LIN {X 0,Y 523.92,Z 267.852,A -85,B 0,C 180,E1 -4812.457,E2 -4812.457} C_VEL
LIN {X 0,Y 523.943,Z 267.84,A -85,B 0,C 180,E1 -4815.311,E2 -4815.311} C_VEL
LIN {X 0,Y 523.959,Z 267.843,A -85,B 0,C 180,E1 -4818.69,E2 -4818.69} C_VEL
LIN {X 0,Y 523.916,Z 267.847,A -85,B 0,C 180,E1 -4821.898,E2 -4821.898} C_VEL
LIN {X 0,Y 523.925,Z 267.843,A -85,B 0,C 180,E1 -4824.912,E2 -4824.912} C_VEL
LIN {X 0,Y 523.939,Z 267.841,A -85,B 0,C 180,E1 -4827.68,E2 -4827.68} C_VEL
LIN {X 0,Y 523.957,Z 267.84,A -85,B 0,C 180,E1 -4830.677,E2 -4830.677} C_VEL
LIN {X 0,Y 523.932,Z 267.843,A -85,B 0,C 180,E1 -4833.726,E2 -4833.726} C_VEL
LIN {X 0,Y 523.915,Z 267.849,A -85,B 0,C 180,E1 -4836.27,E2 -4836.27} C_VEL
LIN {X 0,Y 523.95,Z 267.841,A -85,B 0,C 180,E1 -4838.767,E2 -4838.767} C_VEL
LIN {X 0,Y 523.942,Z 267.839,A -85,B 0,C 180,E1 -4841.22,E2 -4841.22} C_VEL
LIN {X 0,Y 523.926,Z 267.846,A -85,B 0,C 180,E1 -4843.639,E2 -4843.639} C_VEL
LIN {X 0,Y 523.939,Z 267.849,A -85,B 0,C 180,E1 -4846.028,E2 -4846.028} C_VEL
LIN {X 0,Y 523.996,Z 267.832,A -85,B 0,C 180,E1 -4849.177,E2 -4849.177} C_VEL
LIN {X 0,Y 523.96,Z 267.842,A -85,B 0,C 180,E1 -4851.515,E2 -4851.515} C_VEL
LIN {X 0,Y 524.041,Z 267.829,A -85,B 0,C 180,E1 -4854.613,E2 -4854.613} C_VEL
LIN {X 0,Y 524.107,Z 267.825,A -85,B 0,C 180,E1 -4857.695,E2 -4857.695} C_VEL
LIN {X 0,Y 524.1,Z 267.827,A -85,B 0,C 180,E1 -4860,E2 -4860} C_VEL
LIN {X 0,Y 524.037,Z 267.829,A -85,B 0,C 180,E1 -4863.075,E2 -4863.075} C_VEL
LIN {X 0,Y 524.002,Z 267.835,A -85,B 0,C 180,E1 -4866.16,E2 -4866.16} C_VEL
LIN {X 0,Y 523.948,Z 267.843,A -85,B 0,C 180,E1 -4869.263,E2 -4869.263} C_VEL
LIN {X 0,Y 524.001,Z 267.841,A -85,B 0,C 180,E1 -4871.735,E2 -4871.735} C_VEL
LIN {X 0,Y 523.987,Z 267.834,A -85,B 0,C 180,E1 -4875.047,E2 -4875.047} C_VEL
LIN {X 0,Y 523.914,Z 267.846,A -85,B 0,C 180,E1 -4877.971,E2 -4877.971} C_VEL
LIN {X 0,Y 523.92,Z 267.844,A -85,B 0,C 180,E1 -4880.412,E2 -4880.412} C_VEL
LIN {X 0,Y 523.888,Z 267.846,A -85,B 0,C 180,E1 -4882.895,E2 -4882.895} C_VEL
LIN {X 0,Y 523.883,Z 267.856,A -85,B 0,C 180,E1 -4885.422,E2 -4885.422} C_VEL
LIN {X 0,Y 523.9,Z 267.841,A -85,B 0,C 180,E1 -4888.003,E2 -4888.003} C_VEL
LIN {X 0,Y 523.901,Z 267.847,A -85,B 0,C 180,E1 -4890.845,E2 -4890.845} C_VEL
LIN {X 0,Y 523.914,Z 267.849,A -85,B 0,C 180,E1 -4893.726,E2 -4893.726} C_VEL
LIN {X 0,Y 523.86,Z 267.85,A -85,B 0,C 180,E1 -4896.394,E2 -4896.394} C_VEL
LIN {X 0,Y 523.889,Z 267.852,A -85,B 0,C 180,E1 -4899.088,E2 -4899.088} C_VEL
LIN {X 0,Y 523.888,Z 267.847,A -85,B 0,C 180,E1 -4902.125,E2 -4902.125} C_VEL
LIN {X 0,Y 523.927,Z 267.844,A -85,B 0,C 180,E1 -4904.687,E2 -4904.687} C_VEL
LIN {X 0,Y 523.857,Z 267.853,A -85,B 0,C 180,E1 -4906.864,E2 -4906.864} C_VEL
LIN {X 0,Y 523.17,Z 267.942,A -85,B 0,C 180,E1 -4907.506,E2 -4907.506} C_VEL
LIN {X 0,Y 520.306,Z 268.294,A -85,B 0,C 180,E1 -4908.547,E2 -4908.547} C_VEL
LIN {X 0,Y 517.908,Z 268.599,A -85,B 0,C 180,E1 -4909.386,E2 -4909.386} C_VEL
LIN {X 0,Y 516.896,Z 268.719,A -85,B 0,C 180,E1 -4910.034,E2 -4910.034} C_VEL
LIN {X 0,Y 516.822,Z 268.727,A -85,B 0,C 180,E1 -4910.253,E2 -4910.253} C_VEL
LIN {X 0,Y 516.798,Z 268.736,A -85,B 0,C 180,E1 -4913.247,E2 -4913.247} C_VEL
LIN {X 0,Y 516.868,Z 268.721,A -85,B 0,C 180,E1 -4916.117,E2 -4916.117} C_VEL
LIN {X 0,Y 516.85,Z 268.729,A -85,B 0,C 180,E1 -4918.944,E2 -4918.944} C_VEL
LIN {X 0,Y 516.857,Z 268.725,A -85,B 0,C 180,E1 -4922.11,E2 -4922.11} C_VEL
LIN {X 0,Y 516.831,Z 268.735,A -85,B 0,C 180,E1 -4925.067,E2 -4925.067} C_VEL
LIN {X 0,Y 516.903,Z 268.891,A -85,B 0,C 180,E1 -4925.606,E2 -4925.606} C_VEL
LIN {X 0,Y 518.761,Z 277.486,A -85,B 0,C 180,E1 -4927.108,E2 -4927.108} C_VEL
LIN {X 0,Y 518.929,Z 282.515,A -85,B 0,C 180,E1 -4927.924,E2 -4927.924} C_VEL
LIN {X 0,Y 518.898,Z 284.871,A -85,B 0,C 180,E1 -4928.27,E2 -4928.27} C_VEL
LIN {X 0,Y 521.958,Z 298.303,A -85,B 0,C 180,E1 -4928.601,E2 -4928.601} C_VEL
LIN {X 0,Y 520.969,Z 446.051,A -85,B 0,C 180,E1 -4930.702,E2 -4930.702} C_VEL
LIN {X 0,Y 520.739,Z 460.824,A -85,B 0,C 180,E1 -4931.027,E2 -4931.027} C_VEL
LIN {X 0,Y 520.374,Z 475.321,A -85,B 0,C 180,E1 -4931.495,E2 -4931.495} C_VEL
LIN {X 0,Y 519.924,Z 489.139,A -85,B 0,C 180,E1 -4932.09,E2 -4932.09} C_VEL
LIN {X 0,Y 519.531,Z 501.957,A -85,B 0,C 180,E1 -4932.787,E2 -4932.787} C_VEL
LIN {X 0,Y 518.971,Z 515.318,A -85,B 0,C 180,E1 -4933.68,E2 -4933.68} C_VEL
LIN {X 0,Y 518.458,Z 527.648,A -85,B 0,C 180,E1 -4934.682,E2 -4934.682} C_VEL
LIN {X 0,Y 517.945,Z 539.712,A -85,B 0,C 180,E1 -4935.863,E2 -4935.863} C_VEL
LIN {X 0,Y 517.493,Z 549.881,A -85,B 0,C 180,E1 -4937.051,E2 -4937.051} C_VEL
LIN {X 0,Y 517.092,Z 559.832,A -85,B 0,C 180,E1 -4938.435,E2 -4938.435} C_VEL
LIN {X 0,Y 516.786,Z 568.082,A -85,B 0,C 180,E1 -4939.817,E2 -4939.817} C_VEL
LIN {X 0,Y 516.576,Z 575.827,A -85,B 0,C 180,E1 -4941.393,E2 -4941.393} C_VEL
LIN {X 0,Y 516.431,Z 581.994,A -85,B 0,C 180,E1 -4942.964,E2 -4942.964} C_VEL
LIN {X 0,Y 516.377,Z 586.756,A -85,B 0,C 180,E1 -4944.533,E2 -4944.533} C_VEL
LIN {X 0,Y 516.326,Z 590.248,A -85,B 0,C 180,E1 -4946.097,E2 -4946.097} C_VEL
LIN {X 0,Y 516.258,Z 592.562,A -85,B 0,C 180,E1 -4947.659,E2 -4947.659} C_VEL
LIN {X 0,Y 516.156,Z 593.75,A -85,B 0,C 180,E1 -4949.219,E2 -4949.219} C_VEL
LIN {X 0,Y 516.157,Z 593.769,A -85,B 0,C 180,E1 -4950.78,E2 -4950.78} C_VEL
LIN {X 0,Y 516.259,Z 592.657,A -85,B 0,C 180,E1 -4952.34,E2 -4952.34} C_VEL
LIN {X 0,Y 516.326,Z 590.419,A -85,B 0,C 180,E1 -4953.902,E2 -4953.902} C_VEL
LIN {X 0,Y 516.373,Z 586.999,A -85,B 0,C 180,E1 -4955.467,E2 -4955.467} C_VEL
LIN {X 0,Y 516.429,Z 582.315,A -85,B 0,C 180,E1 -4957.035,E2 -4957.035} C_VEL
LIN {X 0,Y 516.573,Z 576.243,A -85,B 0,C 180,E1 -4958.607,E2 -4958.607} C_VEL
LIN {X 0,Y 516.776,Z 568.595,A -85,B 0,C 180,E1 -4960.183,E2 -4960.183} C_VEL
LIN {X 0,Y 517.069,Z 560.435,A -85,B 0,C 180,E1 -4961.565,E2 -4961.565} C_VEL
LIN {X 0,Y 517.471,Z 550.604,A -85,B 0,C 180,E1 -4962.949,E2 -4962.949} C_VEL
LIN {X 0,Y 517.892,Z 540.518,A -85,B 0,C 180,E1 -4964.138,E2 -4964.138} C_VEL
LIN {X 0,Y 518.371,Z 528.692,A -85,B 0,C 180,E1 -4965.312,E2 -4965.312} C_VEL
LIN {X 0,Y 518.996,Z 515.308,A -85,B 0,C 180,E1 -4966.41,E2 -4966.41} C_VEL
LIN {X 0,Y 519.562,Z 501.798,A -85,B 0,C 180,E1 -4967.313,E2 -4967.313} C_VEL
LIN {X 0,Y 520.023,Z 486.91,A -85,B 0,C 180,E1 -4968.11,E2 -4968.11} C_VEL
LIN {X 0,Y 520.477,Z 471.674,A -85,B 0,C 180,E1 -4968.73,E2 -4968.73} C_VEL
LIN {X 0,Y 520.782,Z 456.381,A -85,B 0,C 180,E1 -4969.181,E2 -4969.181} C_VEL
LIN {X 0,Y 521.016,Z 441.647,A -85,B 0,C 180,E1 -4969.46,E2 -4969.46} C_VEL
LIN {X 0,Y 522.012,Z 299.314,A -85,B 0,C 180,E1 -4971.472,E2 -4971.472} C_VEL
LIN {X 0,Y 520.274,Z 290.511,A -85,B 0,C 180,E1 -4971.676,E2 -4971.676} C_VEL
LIN {X 0,Y 518.874,Z 284.647,A -85,B 0,C 180,E1 -4971.83,E2 -4971.83} C_VEL
LIN {X 0,Y 519.035,Z 279.823,A -85,B 0,C 180,E1 -4972.592,E2 -4972.592} C_VEL
LIN {X 0,Y 517.73,Z 272.676,A -85,B 0,C 180,E1 -4973.818,E2 -4973.818} C_VEL
LIN {X 0,Y 516.884,Z 268.728,A -85,B 0,C 180,E1 -4974.516,E2 -4974.516} C_VEL
LIN {X 0,Y 516.867,Z 268.727,A -85,B 0,C 180,E1 -4977.536,E2 -4977.536} C_VEL
LIN {X 0,Y 516.844,Z 268.729,A -85,B 0,C 180,E1 -4980.207,E2 -4980.207} C_VEL
LIN {X 0,Y 516.858,Z 268.731,A -85,B 0,C 180,E1 -4982.949,E2 -4982.949} C_VEL
LIN {X 0,Y 516.817,Z 268.728,A -85,B 0,C 180,E1 -4985.784,E2 -4985.784} C_VEL
LIN {X 0,Y 516.869,Z 268.73,A -85,B 0,C 180,E1 -4988.717,E2 -4988.717} C_VEL
LIN {X 0,Y 516.841,Z 268.726,A -85,B 0,C 180,E1 -4991.782,E2 -4991.782} C_VEL
LIN {X 0,Y 516.894,Z 268.725,A -85,B 0,C 180,E1 -4995.007,E2 -4995.007} C_VEL
LIN {X 0,Y 516.827,Z 268.725,A -85,B 0,C 180,E1 -4998.409,E2 -4998.409} C_VEL
LIN {X 0,Y 516.851,Z 268.725,A -85,B 0,C 180,E1 -5001.281,E2 -5001.281} C_VEL
LIN {X 0,Y 516.824,Z 268.727,A -85,B 0,C 180,E1 -5004.677,E2 -5004.677} C_VEL
LIN {X 0,Y 516.862,Z 268.723,A -85,B 0,C 180,E1 -5007.462,E2 -5007.462} C_VEL
LIN {X 0,Y 516.836,Z 268.733,A -85,B 0,C 180,E1 -5010.491,E2 -5010.491} C_VEL
LIN {X 0,Y 516.83,Z 268.726,A -85,B 0,C 180,E1 -5013.337,E2 -5013.337} C_VEL
LIN {X 0,Y 516.864,Z 268.724,A -85,B 0,C 180,E1 -5015.926,E2 -5015.926} C_VEL
LIN {X 0,Y 516.851,Z 268.732,A -85,B 0,C 180,E1 -5018.461,E2 -5018.461} C_VEL
LIN {X 0,Y 516.872,Z 268.721,A -85,B 0,C 180,E1 -5020.954,E2 -5020.954} C_VEL
LIN {X 0,Y 516.828,Z 268.727,A -85,B 0,C 180,E1 -5023.407,E2 -5023.407} C_VEL
LIN {X 0,Y 516.865,Z 268.722,A -85,B 0,C 180,E1 -5025.833,E2 -5025.833} C_VEL
LIN {X 0,Y 516.942,Z 268.713,A -85,B 0,C 180,E1 -5029.028,E2 -5029.028} C_VEL
LIN {X 0,Y 516.924,Z 268.719,A -85,B 0,C 180,E1 -5032.186,E2 -5032.186} C_VEL
LIN {X 0,Y 516.98,Z 268.711,A -85,B 0,C 180,E1 -5034.539,E2 -5034.539} C_VEL
LIN {X 0,Y 517.074,Z 268.697,A -85,B 0,C 180,E1 -5037.663,E2 -5037.663} C_VEL
LIN {X 0,Y 517.088,Z 268.692,A -85,B 0,C 180,E1 -5040.779,E2 -5040.779} C_VEL
LIN {X 0,Y 516.968,Z 268.709,A -85,B 0,C 180,E1 -5043.117,E2 -5043.117} C_VEL
LIN {X 0,Y 516.972,Z 268.714,A -85,B 0,C 180,E1 -5046.244,E2 -5046.244} C_VEL
LIN {X 0,Y 516.936,Z 268.714,A -85,B 0,C 180,E1 -5049.389,E2 -5049.389} C_VEL
LIN {X 0,Y 516.951,Z 268.714,A -85,B 0,C 180,E1 -5051.807,E2 -5051.807} C_VEL
LIN {X 0,Y 516.944,Z 268.71,A -85,B 0,C 180,E1 -5055.146,E2 -5055.146} C_VEL
LIN {X 0,Y 516.911,Z 268.721,A -85,B 0,C 180,E1 -5058.223,E2 -5058.223} C_VEL
LIN {X 0,Y 516.911,Z 268.717,A -85,B 0,C 180,E1 -5060.701,E2 -5060.701} C_VEL
LIN {X 0,Y 516.889,Z 268.717,A -85,B 0,C 180,E1 -5064.073,E2 -5064.073} C_VEL
LIN {X 0,Y 516.896,Z 268.716,A -85,B 0,C 180,E1 -5066.659,E2 -5066.659} C_VEL
LIN {X 0,Y 516.908,Z 268.722,A -85,B 0,C 180,E1 -5069.523,E2 -5069.523} C_VEL
LIN {X 0,Y 516.894,Z 268.715,A -85,B 0,C 180,E1 -5072.543,E2 -5072.543} C_VEL
LIN {X 0,Y 516.87,Z 268.725,A -85,B 0,C 180,E1 -5075.33,E2 -5075.33} C_VEL
LIN {X 0,Y 516.878,Z 268.723,A -85,B 0,C 180,E1 -5077.943,E2 -5077.943} C_VEL
LIN {X 0,Y 516.881,Z 268.72,A -85,B 0,C 180,E1 -5080.742,E2 -5080.742} C_VEL
LIN {X 0,Y 516.881,Z 268.721,A -85,B 0,C 180,E1 -5082.832,E2 -5082.832} C_VEL
LIN {X 0,Y 516.893,Z 268.72,A -85,B 0,C 180,E1 -5085.007,E2 -5085.007} C_VEL
LIN {X 0,Y 516.912,Z 268.716,A -85,B 0,C 180,E1 -5088.399,E2 -5088.399} C_VEL
LIN {X 0,Y 516.879,Z 268.726,A -85,B 0,C 180,E1 -5091.284,E2 -5091.284} C_VEL
LIN {X 0,Y 516.887,Z 268.722,A -85,B 0,C 180,E1 -5094.221,E2 -5094.221} C_VEL
LIN {X 0,Y 516.894,Z 268.723,A -85,B 0,C 180,E1 -5097.053,E2 -5097.053} C_VEL
LIN {X 0,Y 516.891,Z 268.727,A -85,B 0,C 180,E1 -5099.797,E2 -5099.797} C_VEL
LIN {X 0,Y 516.928,Z 268.855,A -85,B 0,C 180,E1 -5101.281,E2 -5101.281} C_VEL
LIN {X 0,Y 520.068,Z 282.653,A -85,B 0,C 180,E1 -5103.315,E2 -5103.315} C_VEL
LIN {X 0,Y 519.444,Z 305.178,A -85,B 0,C 180,E1 -5106.265,E2 -5106.265} C_VEL
LIN {X 0,Y 518.893,Z 320.181,A -85,B 0,C 180,E1 -5108.197,E2 -5108.197} C_VEL
LIN {X 0,Y 521.904,Z 335.969,A -85,B 0,C 180,E1 -5108.563,E2 -5108.563} C_VEL
LIN {X 0,Y 520.836,Z 485.958,A -85,B 0,C 180,E1 -5110.694,E2 -5110.694} C_VEL
LIN {X 0,Y 520.575,Z 500.684,A -85,B 0,C 180,E1 -5111.042,E2 -5111.042} C_VEL
LIN {X 0,Y 520.166,Z 514.057,A -85,B 0,C 180,E1 -5111.488,E2 -5111.488} C_VEL
LIN {X 0,Y 519.693,Z 527.714,A -85,B 0,C 180,E1 -5112.082,E2 -5112.082} C_VEL
LIN {X 0,Y 519.218,Z 542.063,A -85,B 0,C 180,E1 -5112.879,E2 -5112.879} C_VEL
LIN {X 0,Y 518.679,Z 555.131,A -85,B 0,C 180,E1 -5113.772,E2 -5113.772} C_VEL
LIN {X 0,Y 518.225,Z 566.573,A -85,B 0,C 180,E1 -5114.708,E2 -5114.708} C_VEL
LIN {X 0,Y 517.747,Z 578.379,A -85,B 0,C 180,E1 -5115.858,E2 -5115.858} C_VEL
LIN {X 0,Y 517.359,Z 588.67,A -85,B 0,C 180,E1 -5117.048,E2 -5117.048} C_VEL
LIN {X 0,Y 516.957,Z 598.75,A -85,B 0,C 180,E1 -5118.435,E2 -5118.435} C_VEL
LIN {X 0,Y 516.748,Z 607.095,A -85,B 0,C 180,E1 -5119.817,E2 -5119.817} C_VEL
LIN {X 0,Y 516.515,Z 614.951,A -85,B 0,C 180,E1 -5121.392,E2 -5121.392} C_VEL
LIN {X 0,Y 516.391,Z 621.202,A -85,B 0,C 180,E1 -5122.965,E2 -5122.965} C_VEL
LIN {X 0,Y 516.351,Z 626.04,A -85,B 0,C 180,E1 -5124.533,E2 -5124.533} C_VEL
LIN {X 0,Y 516.307,Z 629.583,A -85,B 0,C 180,E1 -5126.098,E2 -5126.098} C_VEL
LIN {X 0,Y 516.258,Z 631.912,A -85,B 0,C 180,E1 -5127.66,E2 -5127.66} C_VEL
LIN {X 0,Y 516.157,Z 633.082,A -85,B 0,C 180,E1 -5129.22,E2 -5129.22} C_VEL
LIN {X 0,Y 516.157,Z 633.081,A -85,B 0,C 180,E1 -5130.781,E2 -5130.781} C_VEL
LIN {X 0,Y 516.258,Z 631.908,A -85,B 0,C 180,E1 -5132.341,E2 -5132.341} C_VEL
LIN {X 0,Y 516.307,Z 629.577,A -85,B 0,C 180,E1 -5133.903,E2 -5133.903} C_VEL
LIN {X 0,Y 516.351,Z 626.039,A -85,B 0,C 180,E1 -5135.468,E2 -5135.468} C_VEL
LIN {X 0,Y 516.392,Z 621.204,A -85,B 0,C 180,E1 -5137.036,E2 -5137.036} C_VEL
LIN {X 0,Y 516.515,Z 614.944,A -85,B 0,C 180,E1 -5138.608,E2 -5138.608} C_VEL
LIN {X 0,Y 516.749,Z 607.085,A -85,B 0,C 180,E1 -5140.184,E2 -5140.184} C_VEL
LIN {X 0,Y 516.978,Z 598.727,A -85,B 0,C 180,E1 -5141.568,E2 -5141.568} C_VEL
LIN {X 0,Y 517.36,Z 588.664,A -85,B 0,C 180,E1 -5142.953,E2 -5142.953} C_VEL
LIN {X 0,Y 517.724,Z 578.372,A -85,B 0,C 180,E1 -5144.144,E2 -5144.144} C_VEL
LIN {X 0,Y 518.243,Z 566.539,A -85,B 0,C 180,E1 -5145.295,E2 -5145.295} C_VEL
LIN {X 0,Y 518.728,Z 553.828,A -85,B 0,C 180,E1 -5146.328,E2 -5146.328} C_VEL
LIN {X 0,Y 519.3,Z 540.456,A -85,B 0,C 180,E1 -5147.221,E2 -5147.221} C_VEL
LIN {X 0,Y 519.815,Z 525.705,A -85,B 0,C 180,E1 -5148.016,E2 -5148.016} C_VEL
LIN {X 0,Y 520.243,Z 511.445,A -85,B 0,C 180,E1 -5148.612,E2 -5148.612} C_VEL
LIN {X 0,Y 520.629,Z 495.966,A -85,B 0,C 180,E1 -5149.088,E2 -5149.088} C_VEL
LIN {X 0,Y 520.9,Z 480.134,A -85,B 0,C 180,E1 -5149.403,E2 -5149.403} C_VEL
LIN {X 0,Y 521.865,Z 335.63,A -85,B 0,C 180,E1 -5151.443,E2 -5151.443} C_VEL
LIN {X 0,Y 518.918,Z 320.204,A -85,B 0,C 180,E1 -5151.799,E2 -5151.799} C_VEL
LIN {X 0,Y 519.657,Z 297.1,A -85,B 0,C 180,E1 -5154.788,E2 -5154.788} C_VEL
LIN {X 0,Y 520.077,Z 282.636,A -85,B 0,C 180,E1 -5156.686,E2 -5156.686} C_VEL
LIN {X 0,Y 517.049,Z 269.454,A -85,B 0,C 180,E1 -5158.63,E2 -5158.63} C_VEL
LIN {X 0,Y 516.905,Z 268.725,A -85,B 0,C 180,E1 -5158.749,E2 -5158.749} C_VEL
LIN {X 0,Y 516.891,Z 268.723,A -85,B 0,C 180,E1 -5161.11,E2 -5161.11} C_VEL
LIN {X 0,Y 516.91,Z 268.721,A -85,B 0,C 180,E1 -5163.966,E2 -5163.966} C_VEL
LIN {X 0,Y 516.879,Z 268.726,A -85,B 0,C 180,E1 -5166.747,E2 -5166.747} C_VEL
LIN {X 0,Y 516.885,Z 268.718,A -85,B 0,C 180,E1 -5169.722,E2 -5169.722} C_VEL
LIN {X 0,Y 516.909,Z 268.718,A -85,B 0,C 180,E1 -5171.776,E2 -5171.776} C_VEL
LIN {X 0,Y 516.898,Z 268.72,A -85,B 0,C 180,E1 -5175.007,E2 -5175.007} C_VEL
LIN {X 0,Y 516.916,Z 268.725,A -85,B 0,C 180,E1 -5178.399,E2 -5178.399} C_VEL
LIN {X 0,Y 516.88,Z 268.721,A -85,B 0,C 180,E1 -5181.284,E2 -5181.284} C_VEL
LIN {X 0,Y 516.87,Z 268.729,A -85,B 0,C 180,E1 -5184.22,E2 -5184.22} C_VEL
LIN {X 0,Y 516.899,Z 268.717,A -85,B 0,C 180,E1 -5187.053,E2 -5187.053} C_VEL
LIN {X 0,Y 516.896,Z 268.721,A -85,B 0,C 180,E1 -5189.797,E2 -5189.797} C_VEL
LIN {X 0,Y 516.896,Z 268.722,A -85,B 0,C 180,E1 -5192.466,E2 -5192.466} C_VEL
LIN {X 0,Y 516.865,Z 268.722,A -85,B 0,C 180,E1 -5195.07,E2 -5195.07} C_VEL
LIN {X 0,Y 516.874,Z 268.721,A -85,B 0,C 180,E1 -5197.622,E2 -5197.622} C_VEL
LIN {X 0,Y 516.934,Z 268.72,A -85,B 0,C 180,E1 -5200.13,E2 -5200.13} C_VEL
LIN {X 0,Y 516.9,Z 268.72,A -85,B 0,C 180,E1 -5202.595,E2 -5202.595} C_VEL
LIN {X 0,Y 516.948,Z 268.71,A -85,B 0,C 180,E1 -5205.03,E2 -5205.03} C_VEL
LIN {X 0,Y 516.972,Z 268.712,A -85,B 0,C 180,E1 -5208.234,E2 -5208.234} C_VEL
LIN {X 0,Y 516.936,Z 268.716,A -85,B 0,C 180,E1 -5211.399,E2 -5211.399} C_VEL
LIN {X 0,Y 516.992,Z 268.708,A -85,B 0,C 180,E1 -5214.54,E2 -5214.54} C_VEL
LIN {X 0,Y 517.077,Z 268.7,A -85,B 0,C 180,E1 -5217.663,E2 -5217.663} C_VEL
LIN {X 0,Y 517.069,Z 268.703,A -85,B 0,C 180,E1 -5220,E2 -5220} C_VEL
LIN {X 0,Y 517.079,Z 268.697,A -85,B 0,C 180,E1 -5222.337,E2 -5222.337} C_VEL
LIN {X 0,Y 516.985,Z 268.712,A -85,B 0,C 180,E1 -5225.461,E2 -5225.461} C_VEL
LIN {X 0,Y 516.929,Z 268.715,A -85,B 0,C 180,E1 -5228.601,E2 -5228.601} C_VEL
LIN {X 0,Y 516.958,Z 268.718,A -85,B 0,C 180,E1 -5231.807,E2 -5231.807} C_VEL
LIN {X 0,Y 516.94,Z 268.712,A -85,B 0,C 180,E1 -5235.142,E2 -5235.142} C_VEL
LIN {X 0,Y 516.874,Z 268.72,A -85,B 0,C 180,E1 -5238.224,E2 -5238.224} C_VEL
LIN {X 0,Y 516.875,Z 268.721,A -85,B 0,C 180,E1 -5240.703,E2 -5240.703} C_VEL
LIN {X 0,Y 516.844,Z 268.727,A -85,B 0,C 180,E1 -5243.225,E2 -5243.225} C_VEL
LIN {X 0,Y 516.864,Z 268.721,A -85,B 0,C 180,E1 -5246.177,E2 -5246.177} C_VEL
LIN {X 0,Y 516.832,Z 268.719,A -85,B 0,C 180,E1 -5248.421,E2 -5248.421} C_VEL
LIN {X 0,Y 516.851,Z 268.728,A -85,B 0,C 180,E1 -5251.112,E2 -5251.112} C_VEL
LIN {X 0,Y 516.872,Z 268.724,A -85,B 0,C 180,E1 -5253.959,E2 -5253.959} C_VEL
LIN {X 0,Y 516.802,Z 268.73,A -85,B 0,C 180,E1 -5256.752,E2 -5256.752} C_VEL
LIN {X 0,Y 516.825,Z 268.731,A -85,B 0,C 180,E1 -5259.727,E2 -5259.727} C_VEL
LIN {X 0,Y 516.839,Z 268.728,A -85,B 0,C 180,E1 -5262.836,E2 -5262.836} C_VEL
LIN {X 0,Y 516.865,Z 268.727,A -85,B 0,C 180,E1 -5265.003,E2 -5265.003} C_VEL
LIN {X 0,Y 516.825,Z 268.727,A -85,B 0,C 180,E1 -5268.215,E2 -5268.215} C_VEL
LIN {X 0,Y 516.822,Z 268.727,A -85,B 0,C 180,E1 -5270.253,E2 -5270.253} C_VEL
LIN {X 0,Y 516.177,Z 268.814,A -85,B 0,C 180,E1 -5270.903,E2 -5270.903} C_VEL
LIN {X 0,Y 513.323,Z 269.17,A -85,B 0,C 180,E1 -5271.959,E2 -5271.959} C_VEL
LIN {X 0,Y 510.893,Z 269.474,A -85,B 0,C 180,E1 -5272.809,E2 -5272.809} C_VEL
LIN {X 0,Y 509.844,Z 269.603,A -85,B 0,C 180,E1 -5273.465,E2 -5273.465} C_VEL
LIN {X 0,Y 509.757,Z 269.611,A -85,B 0,C 180,E1 -5273.688,E2 -5273.688} C_VEL
LIN {X 0,Y 509.826,Z 269.6,A -85,B 0,C 180,E1 -5276.536,E2 -5276.536} C_VEL
LIN {X 0,Y 509.803,Z 269.61,A -85,B 0,C 180,E1 -5279.331,E2 -5279.331} C_VEL
LIN {X 0,Y 509.824,Z 269.602,A -85,B 0,C 180,E1 -5282.05,E2 -5282.05} C_VEL
LIN {X 0,Y 509.805,Z 269.611,A -85,B 0,C 180,E1 -5285.135,E2 -5285.135} C_VEL
LIN {X 0,Y 509.841,Z 269.786,A -85,B 0,C 180,E1 -5285.353,E2 -5285.353} C_VEL
LIN {X 0,Y 511.984,Z 279.585,A -85,B 0,C 180,E1 -5287.091,E2 -5287.091} C_VEL
LIN {X 0,Y 512.056,Z 284.864,A -85,B 0,C 180,E1 -5287.95,E2 -5287.95} C_VEL
LIN {X 0,Y 515.362,Z 299.506,A -85,B 0,C 180,E1 -5288.327,E2 -5288.327} C_VEL
LIN {X 0,Y 514.338,Z 442.657,A -85,B 0,C 180,E1 -5290.379,E2 -5290.379} C_VEL
LIN {X 0,Y 514.084,Z 458.097,A -85,B 0,C 180,E1 -5290.686,E2 -5290.686} C_VEL
LIN {X 0,Y 513.728,Z 473.016,A -85,B 0,C 180,E1 -5291.143,E2 -5291.143} C_VEL
LIN {X 0,Y 513.286,Z 487.426,A -85,B 0,C 180,E1 -5291.747,E2 -5291.747} C_VEL
LIN {X 0,Y 512.76,Z 502.237,A -85,B 0,C 180,E1 -5292.553,E2 -5292.553} C_VEL
LIN {X 0,Y 512.152,Z 515.598,A -85,B 0,C 180,E1 -5293.456,E2 -5293.456} C_VEL
LIN {X 0,Y 511.582,Z 528.173,A -85,B 0,C 180,E1 -5294.494,E2 -5294.494} C_VEL
LIN {X 0,Y 511.025,Z 539.989,A -85,B 0,C 180,E1 -5295.667,E2 -5295.667} C_VEL
LIN {X 0,Y 510.546,Z 550.158,A -85,B 0,C 180,E1 -5296.871,E2 -5296.871} C_VEL
LIN {X 0,Y 510.1,Z 560.169,A -85,B 0,C 180,E1 -5298.283,E2 -5298.283} C_VEL
LIN {X 0,Y 509.768,Z 568.357,A -85,B 0,C 180,E1 -5299.675,E2 -5299.675} C_VEL
LIN {X 0,Y 509.549,Z 576.101,A -85,B 0,C 180,E1 -5301.273,E2 -5301.273} C_VEL
LIN {X 0,Y 509.369,Z 582.267,A -85,B 0,C 180,E1 -5302.866,E2 -5302.866} C_VEL
LIN {X 0,Y 509.315,Z 587.028,A -85,B 0,C 180,E1 -5304.457,E2 -5304.457} C_VEL
LIN {X 0,Y 509.252,Z 590.519,A -85,B 0,C 180,E1 -5306.043,E2 -5306.043} C_VEL
LIN {X 0,Y 509.187,Z 592.832,A -85,B 0,C 180,E1 -5307.626,E2 -5307.626} C_VEL
LIN {X 0,Y 509.07,Z 594.02,A -85,B 0,C 180,E1 -5309.209,E2 -5309.209} C_VEL
LIN {X 0,Y 509.071,Z 594.039,A -85,B 0,C 180,E1 -5310.791,E2 -5310.791} C_VEL
LIN {X 0,Y 509.187,Z 592.926,A -85,B 0,C 180,E1 -5312.373,E2 -5312.373} C_VEL
LIN {X 0,Y 509.252,Z 590.688,A -85,B 0,C 180,E1 -5313.956,E2 -5313.956} C_VEL
LIN {X 0,Y 509.31,Z 587.267,A -85,B 0,C 180,E1 -5315.543,E2 -5315.543} C_VEL
LIN {X 0,Y 509.367,Z 582.584,A -85,B 0,C 180,E1 -5317.133,E2 -5317.133} C_VEL
LIN {X 0,Y 509.545,Z 576.511,A -85,B 0,C 180,E1 -5318.726,E2 -5318.726} C_VEL
LIN {X 0,Y 509.759,Z 568.863,A -85,B 0,C 180,E1 -5320.325,E2 -5320.325} C_VEL
LIN {X 0,Y 510.077,Z 560.248,A -85,B 0,C 180,E1 -5321.796,E2 -5321.796} C_VEL
LIN {X 0,Y 510.527,Z 550.87,A -85,B 0,C 180,E1 -5323.129,E2 -5323.129} C_VEL
LIN {X 0,Y 510.983,Z 540.784,A -85,B 0,C 180,E1 -5324.333,E2 -5324.333} C_VEL
LIN {X 0,Y 511.491,Z 529.221,A -85,B 0,C 180,E1 -5325.498,E2 -5325.498} C_VEL
LIN {X 0,Y 512.11,Z 516.983,A -85,B 0,C 180,E1 -5326.524,E2 -5326.524} C_VEL
LIN {X 0,Y 512.702,Z 503.634,A -85,B 0,C 180,E1 -5327.449,E2 -5327.449} C_VEL
LIN {X 0,Y 513.132,Z 491.165,A -85,B 0,C 180,E1 -5328.155,E2 -5328.155} C_VEL
LIN {X 0,Y 513.638,Z 476.571,A -85,B 0,C 180,E1 -5328.808,E2 -5328.808} C_VEL
LIN {X 0,Y 513.989,Z 461.55,A -85,B 0,C 180,E1 -5329.309,E2 -5329.309} C_VEL
LIN {X 0,Y 514.262,Z 446.383,A -85,B 0,C 180,E1 -5329.649,E2 -5329.649} C_VEL
LIN {X 0,Y 515.324,Z 310.312,A -85,B 0,C 180,E1 -5331.606,E2 -5331.606} C_VEL
LIN {X 0,Y 515.317,Z 298.876,A -85,B 0,C 180,E1 -5331.775,E2 -5331.775} C_VEL
LIN {X 0,Y 512.054,Z 284.842,A -85,B 0,C 180,E1 -5332.144,E2 -5332.144} C_VEL
LIN {X 0,Y 512.047,Z 279.978,A -85,B 0,C 180,E1 -5332.932,E2 -5332.932} C_VEL
LIN {X 0,Y 509.824,Z 269.608,A -85,B 0,C 180,E1 -5334.79,E2 -5334.79} C_VEL
LIN {X 0,Y 509.818,Z 269.609,A -85,B 0,C 180,E1 -5337.059,E2 -5337.059} C_VEL
LIN {X 0,Y 509.824,Z 269.604,A -85,B 0,C 180,E1 -5339.753,E2 -5339.753} C_VEL
LIN {X 0,Y 509.82,Z 269.609,A -85,B 0,C 180,E1 -5342.764,E2 -5342.764} C_VEL
LIN {X 0,Y 509.795,Z 269.604,A -85,B 0,C 180,E1 -5345.573,E2 -5345.573} C_VEL
LIN {X 0,Y 509.813,Z 269.605,A -85,B 0,C 180,E1 -5348.341,E2 -5348.341} C_VEL
LIN {X 0,Y 509.8,Z 269.604,A -85,B 0,C 180,E1 -5351.431,E2 -5351.431} C_VEL
LIN {X 0,Y 509.833,Z 269.603,A -85,B 0,C 180,E1 -5354.67,E2 -5354.67} C_VEL
LIN {X 0,Y 509.78,Z 269.599,A -85,B 0,C 180,E1 -5357.505,E2 -5357.505} C_VEL
LIN {X 0,Y 509.804,Z 269.61,A -85,B 0,C 180,E1 -5360.644,E2 -5360.644} C_VEL
LIN {X 0,Y 509.755,Z 269.598,A -85,B 0,C 180,E1 -5363.641,E2 -5363.641} C_VEL
LIN {X 0,Y 509.822,Z 269.606,A -85,B 0,C 180,E1 -5366.536,E2 -5366.536} C_VEL
LIN {X 0,Y 509.799,Z 269.603,A -85,B 0,C 180,E1 -5369.331,E2 -5369.331} C_VEL
LIN {X 0,Y 509.82,Z 269.602,A -85,B 0,C 180,E1 -5372.05,E2 -5372.05} C_VEL
LIN {X 0,Y 509.793,Z 269.61,A -85,B 0,C 180,E1 -5374.699,E2 -5374.699} C_VEL
LIN {X 0,Y 509.822,Z 269.598,A -85,B 0,C 180,E1 -5377.459,E2 -5377.459} C_VEL
LIN {X 0,Y 509.831,Z 269.601,A -85,B 0,C 180,E1 -5380.68,E2 -5380.68} C_VEL
LIN {X 0,Y 509.783,Z 269.605,A -85,B 0,C 180,E1 -5383.171,E2 -5383.171} C_VEL
LIN {X 0,Y 509.839,Z 269.596,A -85,B 0,C 180,E1 -5385.633,E2 -5385.633} C_VEL
LIN {X 0,Y 509.906,Z 269.591,A -85,B 0,C 180,E1 -5388.874,E2 -5388.874} C_VEL
LIN {X 0,Y 509.876,Z 269.595,A -85,B 0,C 180,E1 -5392.077,E2 -5392.077} C_VEL
LIN {X 0,Y 509.932,Z 269.59,A -85,B 0,C 180,E1 -5394.464,E2 -5394.464} C_VEL
LIN {X 0,Y 510.044,Z 269.572,A -85,B 0,C 180,E1 -5397.631,E2 -5397.631} C_VEL
LIN {X 0,Y 510.037,Z 269.57,A -85,B 0,C 180,E1 -5400.789,E2 -5400.789} C_VEL
LIN {X 0,Y 509.911,Z 269.589,A -85,B 0,C 180,E1 -5403.16,E2 -5403.16} C_VEL
LIN {X 0,Y 509.919,Z 269.592,A -85,B 0,C 180,E1 -5406.33,E2 -5406.33} C_VEL
LIN {X 0,Y 509.876,Z 269.595,A -85,B 0,C 180,E1 -5409.521,E2 -5409.521} C_VEL
LIN {X 0,Y 509.903,Z 269.594,A -85,B 0,C 180,E1 -5411.932,E2 -5411.932} C_VEL
LIN {X 0,Y 509.893,Z 269.589,A -85,B 0,C 180,E1 -5415.242,E2 -5415.242} C_VEL
LIN {X 0,Y 509.856,Z 269.596,A -85,B 0,C 180,E1 -5418.484,E2 -5418.484} C_VEL
LIN {X 0,Y 509.849,Z 269.597,A -85,B 0,C 180,E1 -5421.002,E2 -5421.002} C_VEL
LIN {X 0,Y 509.82,Z 269.603,A -85,B 0,C 180,E1 -5423.564,E2 -5423.564} C_VEL
LIN {X 0,Y 509.883,Z 269.591,A -85,B 0,C 180,E1 -5426.372,E2 -5426.372} C_VEL
LIN {X 0,Y 509.856,Z 269.602,A -85,B 0,C 180,E1 -5429.751,E2 -5429.751} C_VEL
LIN {X 0,Y 509.872,Z 269.589,A -85,B 0,C 180,E1 -5432.774,E2 -5432.774} C_VEL
LIN {X 0,Y 509.829,Z 269.606,A -85,B 0,C 180,E1 -5435.579,E2 -5435.579} C_VEL
LIN {X 0,Y 509.848,Z 269.596,A -85,B 0,C 180,E1 -5438.338,E2 -5438.338} C_VEL
LIN {X 0,Y 509.853,Z 269.601,A -85,B 0,C 180,E1 -5441.426,E2 -5441.426} C_VEL
LIN {X 0,Y 509.837,Z 269.598,A -85,B 0,C 180,E1 -5444.67,E2 -5444.67} C_VEL
LIN {X 0,Y 509.854,Z 269.597,A -85,B 0,C 180,E1 -5448.104,E2 -5448.104} C_VEL
LIN {X 0,Y 509.844,Z 269.598,A -85,B 0,C 180,E1 -5450.648,E2 -5450.648} C_VEL
LIN {X 0,Y 509.833,Z 269.606,A -85,B 0,C 180,E1 -5453.648,E2 -5453.648} C_VEL
LIN {X 0,Y 509.86,Z 269.597,A -85,B 0,C 180,E1 -5456.539,E2 -5456.539} C_VEL
LIN {X 0,Y 509.844,Z 269.603,A -85,B 0,C 180,E1 -5459.335,E2 -5459.335} C_VEL
LIN {X 0,Y 509.869,Z 269.606,A -85,B 0,C 180,E1 -5460.986,E2 -5460.986} C_VEL
LIN {X 0,Y 513.177,Z 283.903,A -85,B 0,C 180,E1 -5463.132,E2 -5463.132} C_VEL
LIN {X 0,Y 512.966,Z 293.939,A -85,B 0,C 180,E1 -5464.476,E2 -5464.476} C_VEL
LIN {X 0,Y 512.297,Z 312.538,A -85,B 0,C 180,E1 -5466.926,E2 -5466.926} C_VEL
LIN {X 0,Y 512.024,Z 319.943,A -85,B 0,C 180,E1 -5467.895,E2 -5467.895} C_VEL
LIN {X 0,Y 515.282,Z 337.302,A -85,B 0,C 180,E1 -5468.298,E2 -5468.298} C_VEL
LIN {X 0,Y 514.125,Z 487.143,A -85,B 0,C 180,E1 -5470.46,E2 -5470.46} C_VEL
LIN {X 0,Y 513.8,Z 502.258,A -85,B 0,C 180,E1 -5470.836,E2 -5470.836} C_VEL
LIN {X 0,Y 513.361,Z 516.396,A -85,B 0,C 180,E1 -5471.337,E2 -5471.337} C_VEL
LIN {X 0,Y 512.781,Z 531.434,A -85,B 0,C 180,E1 -5472.039,E2 -5472.039} C_VEL
LIN {X 0,Y 512.221,Z 544.966,A -85,B 0,C 180,E1 -5472.843,E2 -5472.843} C_VEL
LIN {X 0,Y 511.669,Z 558.75,A -85,B 0,C 180,E1 -5473.851,E2 -5473.851} C_VEL
LIN {X 0,Y 511.068,Z 571.228,A -85,B 0,C 180,E1 -5474.956,E2 -5474.956} C_VEL
LIN {X 0,Y 510.552,Z 583.473,A -85,B 0,C 180,E1 -5476.264,E2 -5476.264} C_VEL
LIN {X 0,Y 510.085,Z 594.362,A -85,B 0,C 180,E1 -5477.669,E2 -5477.669} C_VEL
LIN {X 0,Y 509.831,Z 603.439,A -85,B 0,C 180,E1 -5479.074,E2 -5479.074} C_VEL
LIN {X 0,Y 509.513,Z 610.964,A -85,B 0,C 180,E1 -5480.473,E2 -5480.473} C_VEL
LIN {X 0,Y 509.368,Z 617.991,A -85,B 0,C 180,E1 -5482.07,E2 -5482.07} C_VEL
LIN {X 0,Y 509.261,Z 623.517,A -85,B 0,C 180,E1 -5483.662,E2 -5483.662} C_VEL
LIN {X 0,Y 509.157,Z 627.693,A -85,B 0,C 180,E1 -5485.25,E2 -5485.25} C_VEL
LIN {X 0,Y 509.188,Z 630.624,A -85,B 0,C 180,E1 -5486.835,E2 -5486.835} C_VEL
LIN {X 0,Y 509.11,Z 632.369,A -85,B 0,C 180,E1 -5488.418,E2 -5488.418} C_VEL
LIN {X 0,Y 509.062,Z 632.966,A -85,B 0,C 180,E1 -5490,E2 -5490} C_VEL
LIN {X 0,Y 509.11,Z 632.366,A -85,B 0,C 180,E1 -5491.582,E2 -5491.582} C_VEL
LIN {X 0,Y 509.188,Z 630.618,A -85,B 0,C 180,E1 -5493.165,E2 -5493.165} C_VEL
LIN {X 0,Y 509.157,Z 627.689,A -85,B 0,C 180,E1 -5494.751,E2 -5494.751} C_VEL
LIN {X 0,Y 509.238,Z 623.517,A -85,B 0,C 180,E1 -5496.339,E2 -5496.339} C_VEL
LIN {X 0,Y 509.369,Z 617.989,A -85,B 0,C 180,E1 -5497.931,E2 -5497.931} C_VEL
LIN {X 0,Y 509.513,Z 610.953,A -85,B 0,C 180,E1 -5499.528,E2 -5499.528} C_VEL
LIN {X 0,Y 509.827,Z 603.431,A -85,B 0,C 180,E1 -5500.927,E2 -5500.927} C_VEL
LIN {X 0,Y 510.083,Z 594.358,A -85,B 0,C 180,E1 -5502.332,E2 -5502.332} C_VEL
LIN {X 0,Y 510.553,Z 583.466,A -85,B 0,C 180,E1 -5503.737,E2 -5503.737} C_VEL
LIN {X 0,Y 511.07,Z 571.225,A -85,B 0,C 180,E1 -5505.044,E2 -5505.044} C_VEL
LIN {X 0,Y 511.673,Z 558.75,A -85,B 0,C 180,E1 -5506.15,E2 -5506.15} C_VEL
LIN {X 0,Y 512.162,Z 546.476,A -85,B 0,C 180,E1 -5507.057,E2 -5507.057} C_VEL
LIN {X 0,Y 512.732,Z 533.232,A -85,B 0,C 180,E1 -5507.861,E2 -5507.861} C_VEL
LIN {X 0,Y 513.19,Z 519.912,A -85,B 0,C 180,E1 -5508.514,E2 -5508.514} C_VEL
LIN {X 0,Y 513.653,Z 505.032,A -85,B 0,C 180,E1 -5509.077,E2 -5509.077} C_VEL
LIN {X 0,Y 514.038,Z 489.84,A -85,B 0,C 180,E1 -5509.483,E2 -5509.483} C_VEL
LIN {X 0,Y 514.275,Z 468.193,A -85,B 0,C 180,E1 -5509.835,E2 -5509.835} C_VEL
LIN {X 0,Y 515.305,Z 337.248,A -85,B 0,C 180,E1 -5511.702,E2 -5511.702} C_VEL
LIN {X 0,Y 512.021,Z 319.764,A -85,B 0,C 180,E1 -5512.129,E2 -5512.129} C_VEL
LIN {X 0,Y 512.817,Z 298.461,A -85,B 0,C 180,E1 -5514.925,E2 -5514.925} C_VEL
LIN {X 0,Y 513.31,Z 285.516,A -85,B 0,C 180,E1 -5516.641,E2 -5516.641} C_VEL
LIN {X 0,Y 512.515,Z 280.554,A -85,B 0,C 180,E1 -5517.357,E2 -5517.357} C_VEL
LIN {X 0,Y 509.869,Z 269.601,A -85,B 0,C 180,E1 -5519.014,E2 -5519.014} C_VEL
LIN {X 0,Y 509.822,Z 269.602,A -85,B 0,C 180,E1 -5521.591,E2 -5521.591} C_VEL
LIN {X 0,Y 509.85,Z 269.604,A -85,B 0,C 180,E1 -5524.414,E2 -5524.414} C_VEL
LIN {X 0,Y 509.819,Z 269.601,A -85,B 0,C 180,E1 -5527.341,E2 -5527.341} C_VEL
LIN {X 0,Y 509.84,Z 269.601,A -85,B 0,C 180,E1 -5530.383,E2 -5530.383} C_VEL
LIN {X 0,Y 509.803,Z 269.603,A -85,B 0,C 180,E1 -5533.06,E2 -5533.06} C_VEL
LIN {X 0,Y 509.825,Z 269.601,A -85,B 0,C 180,E1 -5535.794,E2 -5535.794} C_VEL
LIN {X 0,Y 509.858,Z 269.601,A -85,B 0,C 180,E1 -5538.575,E2 -5538.575} C_VEL
LIN {X 0,Y 509.853,Z 269.598,A -85,B 0,C 180,E1 -5541.787,E2 -5541.787} C_VEL
LIN {X 0,Y 509.83,Z 269.601,A -85,B 0,C 180,E1 -5544.622,E2 -5544.622} C_VEL
LIN {X 0,Y 509.865,Z 269.593,A -85,B 0,C 180,E1 -5547.481,E2 -5547.481} C_VEL
LIN {X 0,Y 509.863,Z 269.599,A -85,B 0,C 180,E1 -5550.274,E2 -5550.274} C_VEL
LIN {X 0,Y 509.856,Z 269.594,A -85,B 0,C 180,E1 -5552.943,E2 -5552.943} C_VEL
LIN {X 0,Y 509.849,Z 269.597,A -85,B 0,C 180,E1 -5555.573,E2 -5555.573} C_VEL
LIN {X 0,Y 509.827,Z 269.606,A -85,B 0,C 180,E1 -5558.149,E2 -5558.149} C_VEL
LIN {X 0,Y 509.861,Z 269.594,A -85,B 0,C 180,E1 -5560.682,E2 -5560.682} C_VEL
LIN {X 0,Y 509.869,Z 269.594,A -85,B 0,C 180,E1 -5563.174,E2 -5563.174} C_VEL
LIN {X 0,Y 509.866,Z 269.596,A -85,B 0,C 180,E1 -5565.634,E2 -5565.634} C_VEL
LIN {X 0,Y 509.916,Z 269.585,A -85,B 0,C 180,E1 -5568.875,E2 -5568.875} C_VEL
LIN {X 0,Y 509.882,Z 269.596,A -85,B 0,C 180,E1 -5572.077,E2 -5572.077} C_VEL
LIN {X 0,Y 509.946,Z 269.586,A -85,B 0,C 180,E1 -5574.464,E2 -5574.464} C_VEL
LIN {X 0,Y 510.046,Z 269.575,A -85,B 0,C 180,E1 -5577.631,E2 -5577.631} C_VEL
LIN {X 0,Y 510.038,Z 269.578,A -85,B 0,C 180,E1 -5580,E2 -5580} C_VEL
LIN {X 0,Y 510.05,Z 269.572,A -85,B 0,C 180,E1 -5582.369,E2 -5582.369} C_VEL
LIN {X 0,Y 509.938,Z 269.59,A -85,B 0,C 180,E1 -5585.536,E2 -5585.536} C_VEL
LIN {X 0,Y 509.882,Z 269.599,A -85,B 0,C 180,E1 -5587.923,E2 -5587.923} C_VEL
LIN {X 0,Y 509.912,Z 269.587,A -85,B 0,C 180,E1 -5591.126,E2 -5591.126} C_VEL
LIN {X 0,Y 509.845,Z 269.595,A -85,B 0,C 180,E1 -5594.367,E2 -5594.367} C_VEL
LIN {X 0,Y 509.8,Z 269.603,A -85,B 0,C 180,E1 -5596.828,E2 -5596.828} C_VEL
LIN {X 0,Y 509.83,Z 269.601,A -85,B 0,C 180,E1 -5599.32,E2 -5599.32} C_VEL
LIN {X 0,Y 509.828,Z 269.597,A -85,B 0,C 180,E1 -5602.541,E2 -5602.541} C_VEL
LIN {X 0,Y 509.79,Z 269.61,A -85,B 0,C 180,E1 -5605.301,E2 -5605.301} C_VEL
LIN {X 0,Y 509.811,Z 269.595,A -85,B 0,C 180,E1 -5608.081,E2 -5608.081} C_VEL
LIN {X 0,Y 509.818,Z 269.606,A -85,B 0,C 180,E1 -5611.274,E2 -5611.274} C_VEL
LIN {X 0,Y 509.824,Z 269.6,A -85,B 0,C 180,E1 -5614.416,E2 -5614.416} C_VEL
LIN {X 0,Y 509.766,Z 269.614,A -85,B 0,C 180,E1 -5617.345,E2 -5617.345} C_VEL
LIN {X 0,Y 509.788,Z 269.604,A -85,B 0,C 180,E1 -5620.387,E2 -5620.387} C_VEL
LIN {X 0,Y 509.793,Z 269.608,A -85,B 0,C 180,E1 -5623.575,E2 -5623.575} C_VEL
LIN {X 0,Y 509.773,Z 269.605,A -85,B 0,C 180,E1 -5626.423,E2 -5626.423} C_VEL
LIN {X 0,Y 509.787,Z 269.607,A -85,B 0,C 180,E1 -5629.612,E2 -5629.612} C_VEL
LIN {X 0,Y 509.76,Z 269.609,A -85,B 0,C 180,E1 -5632.654,E2 -5632.654} C_VEL
LIN {X 0,Y 509.757,Z 269.611,A -85,B 0,C 180,E1 -5633.688,E2 -5633.688} C_VEL
LIN {X 0,Y 509.095,Z 269.693,A -85,B 0,C 180,E1 -5634.348,E2 -5634.348} C_VEL
LIN {X 0,Y 506.278,Z 270.047,A -85,B 0,C 180,E1 -5635.42,E2 -5635.42} C_VEL
LIN {X 0,Y 503.89,Z 270.347,A -85,B 0,C 180,E1 -5636.284,E2 -5636.284} C_VEL
LIN {X 0,Y 502.851,Z 270.474,A -85,B 0,C 180,E1 -5636.951,E2 -5636.951} C_VEL
LIN {X 0,Y 502.759,Z 270.483,A -85,B 0,C 180,E1 -5637.177,E2 -5637.177} C_VEL
LIN {X 0,Y 502.745,Z 270.484,A -85,B 0,C 180,E1 -5640.079,E2 -5640.079} C_VEL
LIN {X 0,Y 502.77,Z 270.482,A -85,B 0,C 180,E1 -5642.529,E2 -5642.529} C_VEL
LIN {X 0,Y 502.784,Z 270.531,A -85,B 0,C 180,E1 -5645.068,E2 -5645.068} C_VEL
LIN {X 0,Y 505.179,Z 281.713,A -85,B 0,C 180,E1 -5647.074,E2 -5647.074} C_VEL
LIN {X 0,Y 505.229,Z 285.131,A -85,B 0,C 180,E1 -5647.637,E2 -5647.637} C_VEL
LIN {X 0,Y 508.735,Z 299.898,A -85,B 0,C 180,E1 -5648.031,E2 -5648.031} C_VEL
LIN {X 0,Y 507.93,Z 413.373,A -85,B 0,C 180,E1 -5649.683,E2 -5649.683} C_VEL
LIN {X 0,Y 507.539,Z 451.234,A -85,B 0,C 180,E1 -5650.258,E2 -5650.258} C_VEL
LIN {X 0,Y 507.224,Z 466.529,A -85,B 0,C 180,E1 -5650.655,E2 -5650.655} C_VEL
LIN {X 0,Y 506.796,Z 480.984,A -85,B 0,C 180,E1 -5651.19,E2 -5651.19} C_VEL
LIN {X 0,Y 506.274,Z 495.554,A -85,B 0,C 180,E1 -5651.904,E2 -5651.904} C_VEL
LIN {X 0,Y 505.65,Z 508.806,A -85,B 0,C 180,E1 -5652.717,E2 -5652.717} C_VEL
LIN {X 0,Y 505.093,Z 521.269,A -85,B 0,C 180,E1 -5653.655,E2 -5653.655} C_VEL
LIN {X 0,Y 504.481,Z 533.421,A -85,B 0,C 180,E1 -5654.754,E2 -5654.754} C_VEL
LIN {X 0,Y 503.928,Z 543.808,A -85,B 0,C 180,E1 -5655.873,E2 -5655.873} C_VEL
LIN {X 0,Y 503.453,Z 553.437,A -85,B 0,C 180,E1 -5657.093,E2 -5657.093} C_VEL
LIN {X 0,Y 503.024,Z 563.016,A -85,B 0,C 180,E1 -5658.54,E2 -5658.54} C_VEL
LIN {X 0,Y 502.715,Z 570.72,A -85,B 0,C 180,E1 -5659.935,E2 -5659.935} C_VEL
LIN {X 0,Y 502.465,Z 578.047,A -85,B 0,C 180,E1 -5661.554,E2 -5661.554} C_VEL
LIN {X 0,Y 502.256,Z 583.984,A -85,B 0,C 180,E1 -5663.209,E2 -5663.209} C_VEL
LIN {X 0,Y 502.256,Z 587.299,A -85,B 0,C 180,E1 -5664.378,E2 -5664.378} C_VEL
LIN {X 0,Y 502.181,Z 590.79,A -85,B 0,C 180,E1 -5665.987,E2 -5665.987} C_VEL
LIN {X 0,Y 502.117,Z 593.102,A -85,B 0,C 180,E1 -5667.593,E2 -5667.593} C_VEL
LIN {X 0,Y 501.987,Z 594.29,A -85,B 0,C 180,E1 -5669.197,E2 -5669.197} C_VEL
LIN {X 0,Y 501.988,Z 594.309,A -85,B 0,C 180,E1 -5670.802,E2 -5670.802} C_VEL
LIN {X 0,Y 502.118,Z 593.195,A -85,B 0,C 180,E1 -5672.406,E2 -5672.406} C_VEL
LIN {X 0,Y 502.181,Z 590.957,A -85,B 0,C 180,E1 -5674.012,E2 -5674.012} C_VEL
LIN {X 0,Y 502.249,Z 587.536,A -85,B 0,C 180,E1 -5675.621,E2 -5675.621} C_VEL
LIN {X 0,Y 502.31,Z 582.853,A -85,B 0,C 180,E1 -5677.234,E2 -5677.234} C_VEL
LIN {X 0,Y 502.492,Z 576.78,A -85,B 0,C 180,E1 -5678.85,E2 -5678.85} C_VEL
LIN {X 0,Y 502.747,Z 569.131,A -85,B 0,C 180,E1 -5680.47,E2 -5680.47} C_VEL
LIN {X 0,Y 503.085,Z 560.928,A -85,B 0,C 180,E1 -5681.898,E2 -5681.898} C_VEL
LIN {X 0,Y 503.604,Z 551.136,A -85,B 0,C 180,E1 -5683.312,E2 -5683.312} C_VEL
LIN {X 0,Y 504.089,Z 541.05,A -85,B 0,C 180,E1 -5684.534,E2 -5684.534} C_VEL
LIN {X 0,Y 504.625,Z 529.756,A -85,B 0,C 180,E1 -5685.688,E2 -5685.688} C_VEL
LIN {X 0,Y 505.292,Z 517.246,A -85,B 0,C 180,E1 -5686.753,E2 -5686.753} C_VEL
LIN {X 0,Y 505.925,Z 503.895,A -85,B 0,C 180,E1 -5687.69,E2 -5687.69} C_VEL
LIN {X 0,Y 506.392,Z 491.423,A -85,B 0,C 180,E1 -5688.405,E2 -5688.405} C_VEL
LIN {X 0,Y 506.94,Z 476.824,A -85,B 0,C 180,E1 -5689.066,E2 -5689.066} C_VEL
LIN {X 0,Y 507.32,Z 461.157,A -85,B 0,C 180,E1 -5689.592,E2 -5689.592} C_VEL
LIN {X 0,Y 507.626,Z 445.846,A -85,B 0,C 180,E1 -5689.931,E2 -5689.931} C_VEL
LIN {X 0,Y 508.732,Z 312.404,A -85,B 0,C 180,E1 -5691.872,E2 -5691.872} C_VEL
LIN {X 0,Y 508.734,Z 300.026,A -85,B 0,C 180,E1 -5692.057,E2 -5692.057} C_VEL
LIN {X 0,Y 505.282,Z 285.138,A -85,B 0,C 180,E1 -5692.45,E2 -5692.45} C_VEL
LIN {X 0,Y 505.109,Z 281.165,A -85,B 0,C 180,E1 -5693.111,E2 -5693.111} C_VEL
LIN {X 0,Y 502.774,Z 270.486,A -85,B 0,C 180,E1 -5695.069,E2 -5695.069} C_VEL
LIN {X 0,Y 502.771,Z 270.484,A -85,B 0,C 180,E1 -5697.47,E2 -5697.47} C_VEL
LIN {X 0,Y 502.78,Z 270.482,A -85,B 0,C 180,E1 -5700.213,E2 -5700.213} C_VEL
LIN {X 0,Y 502.768,Z 270.486,A -85,B 0,C 180,E1 -5703.036,E2 -5703.036} C_VEL
LIN {X 0,Y 502.745,Z 270.481,A -85,B 0,C 180,E1 -5705.953,E2 -5705.953} C_VEL
LIN {X 0,Y 502.78,Z 270.485,A -85,B 0,C 180,E1 -5708.978,E2 -5708.978} C_VEL
LIN {X 0,Y 502.743,Z 270.483,A -85,B 0,C 180,E1 -5712.191,E2 -5712.191} C_VEL
LIN {X 0,Y 502.776,Z 270.479,A -85,B 0,C 180,E1 -5715.471,E2 -5715.471} C_VEL
LIN {X 0,Y 502.747,Z 270.485,A -85,B 0,C 180,E1 -5718.927,E2 -5718.927} C_VEL
LIN {X 0,Y 502.744,Z 270.482,A -85,B 0,C 180,E1 -5722.042,E2 -5722.042} C_VEL
LIN {X 0,Y 502.765,Z 270.481,A -85,B 0,C 180,E1 -5725.031,E2 -5725.031} C_VEL
LIN {X 0,Y 502.754,Z 270.481,A -85,B 0,C 180,E1 -5727.913,E2 -5727.913} C_VEL
LIN {X 0,Y 502.75,Z 270.487,A -85,B 0,C 180,E1 -5730.707,E2 -5730.707} C_VEL
LIN {X 0,Y 502.77,Z 270.478,A -85,B 0,C 180,E1 -5733.46,E2 -5733.46} C_VEL
LIN {X 0,Y 502.75,Z 270.483,A -85,B 0,C 180,E1 -5736.084,E2 -5736.084} C_VEL
LIN {X 0,Y 502.757,Z 270.486,A -85,B 0,C 180,E1 -5738.688,E2 -5738.688} C_VEL
LIN {X 0,Y 502.792,Z 270.474,A -85,B 0,C 180,E1 -5741.896,E2 -5741.896} C_VEL
LIN {X 0,Y 502.834,Z 270.473,A -85,B 0,C 180,E1 -5744.665,E2 -5744.665} C_VEL
LIN {X 0,Y 502.876,Z 270.469,A -85,B 0,C 180,E1 -5748.039,E2 -5748.039} C_VEL
LIN {X 0,Y 502.84,Z 270.466,A -85,B 0,C 180,E1 -5751.156,E2 -5751.156} C_VEL
LIN {X 0,Y 502.848,Z 270.469,A -85,B 0,C 180,E1 -5753.58,E2 -5753.58} C_VEL
LIN {X 0,Y 502.864,Z 270.467,A -85,B 0,C 180,E1 -5756.795,E2 -5756.795} C_VEL
LIN {X 0,Y 502.897,Z 270.469,A -85,B 0,C 180,E1 -5758.398,E2 -5758.398} C_VEL
LIN {X 0,Y 502.988,Z 270.448,A -85,B 0,C 180,E1 -5760.801,E2 -5760.801} C_VEL
LIN {X 0,Y 503.012,Z 270.454,A -85,B 0,C 180,E1 -5762.402,E2 -5762.402} C_VEL
LIN {X 0,Y 502.914,Z 270.46,A -85,B 0,C 180,E1 -5765.614,E2 -5765.614} C_VEL
LIN {X 0,Y 502.859,Z 270.467,A -85,B 0,C 180,E1 -5768.843,E2 -5768.843} C_VEL
LIN {X 0,Y 502.844,Z 270.476,A -85,B 0,C 180,E1 -5772.102,E2 -5772.102} C_VEL
LIN {X 0,Y 502.848,Z 270.467,A -85,B 0,C 180,E1 -5775.4,E2 -5775.4} C_VEL
LIN {X 0,Y 502.821,Z 270.471,A -85,B 0,C 180,E1 -5778.752,E2 -5778.752} C_VEL
LIN {X 0,Y 502.782,Z 270.479,A -85,B 0,C 180,E1 -5781.311,E2 -5781.311} C_VEL
LIN {X 0,Y 502.773,Z 270.477,A -85,B 0,C 180,E1 -5783.915,E2 -5783.915} C_VEL
LIN {X 0,Y 502.834,Z 270.468,A -85,B 0,C 180,E1 -5786.568,E2 -5786.568} C_VEL
LIN {X 0,Y 502.813,Z 270.476,A -85,B 0,C 180,E1 -5789.935,E2 -5789.935} C_VEL
LIN {X 0,Y 502.83,Z 270.466,A -85,B 0,C 180,E1 -5793.031,E2 -5793.031} C_VEL
LIN {X 0,Y 502.774,Z 270.48,A -85,B 0,C 180,E1 -5795.951,E2 -5795.951} C_VEL
LIN {X 0,Y 502.799,Z 270.474,A -85,B 0,C 180,E1 -5798.976,E2 -5798.976} C_VEL
LIN {X 0,Y 502.793,Z 270.478,A -85,B 0,C 180,E1 -5802.14,E2 -5802.14} C_VEL
LIN {X 0,Y 502.784,Z 270.482,A -85,B 0,C 180,E1 -5805.47,E2 -5805.47} C_VEL
LIN {X 0,Y 502.818,Z 270.472,A -85,B 0,C 180,E1 -5808.934,E2 -5808.934} C_VEL
LIN {X 0,Y 502.792,Z 270.478,A -85,B 0,C 180,E1 -5812.046,E2 -5812.046} C_VEL
LIN {X 0,Y 502.806,Z 270.479,A -85,B 0,C 180,E1 -5815.035,E2 -5815.035} C_VEL
LIN {X 0,Y 502.782,Z 270.481,A -85,B 0,C 180,E1 -5817.916,E2 -5817.916} C_VEL
LIN {X 0,Y 502.883,Z 270.563,A -85,B 0,C 180,E1 -5820.716,E2 -5820.716} C_VEL
LIN {X 0,Y 506.244,Z 284.934,A -85,B 0,C 180,E1 -5822.912,E2 -5822.912} C_VEL
LIN {X 0,Y 506.354,Z 290.126,A -85,B 0,C 180,E1 -5823.632,E2 -5823.632} C_VEL
LIN {X 0,Y 505.547,Z 310.828,A -85,B 0,C 180,E1 -5826.404,E2 -5826.404} C_VEL
LIN {X 0,Y 505.177,Z 319.625,A -85,B 0,C 180,E1 -5827.573,E2 -5827.573} C_VEL
LIN {X 0,Y 508.693,Z 338.891,A -85,B 0,C 180,E1 -5828.03,E2 -5828.03} C_VEL
LIN {X 0,Y 507.442,Z 486.236,A -85,B 0,C 180,E1 -5830.178,E2 -5830.178} C_VEL
LIN {X 0,Y 507.102,Z 501.348,A -85,B 0,C 180,E1 -5830.553,E2 -5830.553} C_VEL
LIN {X 0,Y 506.594,Z 516.433,A -85,B 0,C 180,E1 -5831.091,E2 -5831.091} C_VEL
LIN {X 0,Y 505.999,Z 531.162,A -85,B 0,C 180,E1 -5831.79,E2 -5831.79} C_VEL
LIN {X 0,Y 505.395,Z 544.693,A -85,B 0,C 180,E1 -5832.604,E2 -5832.604} C_VEL
LIN {X 0,Y 504.807,Z 557.177,A -85,B 0,C 180,E1 -5833.521,E2 -5833.521} C_VEL
LIN {X 0,Y 504.271,Z 568.354,A -85,B 0,C 180,E1 -5834.499,E2 -5834.499} C_VEL
LIN {X 0,Y 503.724,Z 579.627,A -85,B 0,C 180,E1 -5835.662,E2 -5835.662} C_VEL
LIN {X 0,Y 503.299,Z 589.647,A -85,B 0,C 180,E1 -5836.885,E2 -5836.885} C_VEL
LIN {X 0,Y 502.862,Z 598.749,A -85,B 0,C 180,E1 -5838.193,E2 -5838.193} C_VEL
LIN {X 0,Y 502.636,Z 606.549,A -85,B 0,C 180,E1 -5839.527,E2 -5839.527} C_VEL
LIN {X 0,Y 502.353,Z 614.405,A -85,B 0,C 180,E1 -5841.148,E2 -5841.148} C_VEL
LIN {X 0,Y 502.238,Z 620.659,A -85,B 0,C 180,E1 -5842.765,E2 -5842.765} C_VEL
LIN {X 0,Y 502.173,Z 625.497,A -85,B 0,C 180,E1 -5844.378,E2 -5844.378} C_VEL
LIN {X 0,Y 502.095,Z 629.04,A -85,B 0,C 180,E1 -5845.987,E2 -5845.987} C_VEL
LIN {X 0,Y 502.088,Z 631.372,A -85,B 0,C 180,E1 -5847.594,E2 -5847.594} C_VEL
LIN {X 0,Y 501.988,Z 632.542,A -85,B 0,C 180,E1 -5849.198,E2 -5849.198} C_VEL
LIN {X 0,Y 501.988,Z 632.541,A -85,B 0,C 180,E1 -5850.803,E2 -5850.803} C_VEL
LIN {X 0,Y 502.088,Z 631.367,A -85,B 0,C 180,E1 -5852.407,E2 -5852.407} C_VEL
LIN {X 0,Y 502.095,Z 629.034,A -85,B 0,C 180,E1 -5854.014,E2 -5854.014} C_VEL
LIN {X 0,Y 502.171,Z 625.496,A -85,B 0,C 180,E1 -5855.622,E2 -5855.622} C_VEL
LIN {X 0,Y 502.239,Z 620.66,A -85,B 0,C 180,E1 -5857.235,E2 -5857.235} C_VEL
LIN {X 0,Y 502.354,Z 614.398,A -85,B 0,C 180,E1 -5858.853,E2 -5858.853} C_VEL
LIN {X 0,Y 502.636,Z 606.538,A -85,B 0,C 180,E1 -5860.473,E2 -5860.473} C_VEL
LIN {X 0,Y 502.931,Z 597.551,A -85,B 0,C 180,E1 -5861.99,E2 -5861.99} C_VEL
LIN {X 0,Y 503.352,Z 588.116,A -85,B 0,C 180,E1 -5863.32,E2 -5863.32} C_VEL
LIN {X 0,Y 503.792,Z 577.825,A -85,B 0,C 180,E1 -5864.543,E2 -5864.543} C_VEL
LIN {X 0,Y 504.413,Z 565.66,A -85,B 0,C 180,E1 -5865.757,E2 -5865.757} C_VEL
LIN {X 0,Y 505.041,Z 551.939,A -85,B 0,C 180,E1 -5866.888,E2 -5866.888} C_VEL
LIN {X 0,Y 505.749,Z 538.281,A -85,B 0,C 180,E1 -5867.802,E2 -5867.802} C_VEL
LIN {X 0,Y 506.282,Z 524.136,A -85,B 0,C 180,E1 -5868.567,E2 -5868.567} C_VEL
LIN {X 0,Y 506.843,Z 508.617,A -85,B 0,C 180,E1 -5869.21,E2 -5869.21} C_VEL
LIN {X 0,Y 507.269,Z 493.688,A -85,B 0,C 180,E1 -5869.658,E2 -5869.658} C_VEL
LIN {X 0,Y 507.518,Z 477.774,A -85,B 0,C 180,E1 -5869.965,E2 -5869.965} C_VEL
LIN {X 0,Y 508.694,Z 338.349,A -85,B 0,C 180,E1 -5871.978,E2 -5871.978} C_VEL
LIN {X 0,Y 505.203,Z 319.491,A -85,B 0,C 180,E1 -5872.444,E2 -5872.444} C_VEL
LIN {X 0,Y 506.061,Z 297.695,A -85,B 0,C 180,E1 -5875.349,E2 -5875.349} C_VEL
LIN {X 0,Y 506.475,Z 286.877,A -85,B 0,C 180,E1 -5876.807,E2 -5876.807} C_VEL
LIN {X 0,Y 505.605,Z 281.983,A -85,B 0,C 180,E1 -5877.528,E2 -5877.528} C_VEL
LIN {X 0,Y 502.864,Z 270.471,A -85,B 0,C 180,E1 -5879.311,E2 -5879.311} C_VEL
LIN {X 0,Y 502.785,Z 270.481,A -85,B 0,C 180,E1 -5882.085,E2 -5882.085} C_VEL
LIN {X 0,Y 502.801,Z 270.479,A -85,B 0,C 180,E1 -5884.966,E2 -5884.966} C_VEL
LIN {X 0,Y 502.795,Z 270.478,A -85,B 0,C 180,E1 -5887.954,E2 -5887.954} C_VEL
LIN {X 0,Y 502.802,Z 270.476,A -85,B 0,C 180,E1 -5891.068,E2 -5891.068} C_VEL
LIN {X 0,Y 502.782,Z 270.484,A -85,B 0,C 180,E1 -5894.34,E2 -5894.34} C_VEL
LIN {X 0,Y 502.775,Z 270.479,A -85,B 0,C 180,E1 -5896.769,E2 -5896.769} C_VEL
LIN {X 0,Y 502.822,Z 270.473,A -85,B 0,C 180,E1 -5899.006,E2 -5899.006} C_VEL
LIN {X 0,Y 502.793,Z 270.481,A -85,B 0,C 180,E1 -5902.046,E2 -5902.046} C_VEL
LIN {X 0,Y 502.8,Z 270.473,A -85,B 0,C 180,E1 -5905.034,E2 -5905.034} C_VEL
LIN {X 0,Y 502.788,Z 270.478,A -85,B 0,C 180,E1 -5907.916,E2 -5907.916} C_VEL
LIN {X 0,Y 502.817,Z 270.472,A -85,B 0,C 180,E1 -5910.712,E2 -5910.712} C_VEL
LIN {X 0,Y 502.805,Z 270.473,A -85,B 0,C 180,E1 -5913.454,E2 -5913.454} C_VEL
LIN {X 0,Y 502.777,Z 270.484,A -85,B 0,C 180,E1 -5916.086,E2 -5916.086} C_VEL
LIN {X 0,Y 502.786,Z 270.478,A -85,B 0,C 180,E1 -5918.689,E2 -5918.689} C_VEL
LIN {X 0,Y 502.827,Z 270.469,A -85,B 0,C 180,E1 -5921.248,E2 -5921.248} C_VEL
LIN {X 0,Y 502.854,Z 270.467,A -85,B 0,C 180,E1 -5924.601,E2 -5924.601} C_VEL
LIN {X 0,Y 502.882,Z 270.469,A -85,B 0,C 180,E1 -5928.039,E2 -5928.039} C_VEL
LIN {X 0,Y 502.854,Z 270.468,A -85,B 0,C 180,E1 -5931.156,E2 -5931.156} C_VEL
LIN {X 0,Y 502.875,Z 270.466,A -85,B 0,C 180,E1 -5933.581,E2 -5933.581} C_VEL
LIN {X 0,Y 502.84,Z 270.467,A -85,B 0,C 180,E1 -5936.795,E2 -5936.795} C_VEL
LIN {X 0,Y 502.896,Z 270.464,A -85,B 0,C 180,E1 -5938.398,E2 -5938.398} C_VEL
LIN {X 0,Y 503.007,Z 270.454,A -85,B 0,C 180,E1 -5940,E2 -5940} C_VEL
LIN {X 0,Y 503.019,Z 270.448,A -85,B 0,C 180,E1 -5942.402,E2 -5942.402} C_VEL
LIN {X 0,Y 502.893,Z 270.469,A -85,B 0,C 180,E1 -5945.614,E2 -5945.614} C_VEL
LIN {X 0,Y 502.853,Z 270.473,A -85,B 0,C 180,E1 -5948.034,E2 -5948.034} C_VEL
LIN {X 0,Y 502.878,Z 270.465,A -85,B 0,C 180,E1 -5951.283,E2 -5951.283} C_VEL
LIN {X 0,Y 502.827,Z 270.468,A -85,B 0,C 180,E1 -5954.571,E2 -5954.571} C_VEL
LIN {X 0,Y 502.789,Z 270.478,A -85,B 0,C 180,E1 -5957.91,E2 -5957.91} C_VEL
LIN {X 0,Y 502.807,Z 270.474,A -85,B 0,C 180,E1 -5960.527,E2 -5960.527} C_VEL
LIN {X 0,Y 502.783,Z 270.476,A -85,B 0,C 180,E1 -5963.041,E2 -5963.041} C_VEL
LIN {X 0,Y 502.766,Z 270.482,A -85,B 0,C 180,E1 -5965.68,E2 -5965.68} C_VEL
LIN {X 0,Y 502.763,Z 270.471,A -85,B 0,C 180,E1 -5968.378,E2 -5968.378} C_VEL
LIN {X 0,Y 502.768,Z 270.486,A -85,B 0,C 180,E1 -5971.493,E2 -5971.493} C_VEL
LIN {X 0,Y 502.776,Z 270.478,A -85,B 0,C 180,E1 -5974.439,E2 -5974.439} C_VEL
LIN {X 0,Y 502.722,Z 270.489,A -85,B 0,C 180,E1 -5977.168,E2 -5977.168} C_VEL
LIN {X 0,Y 502.732,Z 270.484,A -85,B 0,C 180,E1 -5980.021,E2 -5980.021} C_VEL
LIN {X 0,Y 502.74,Z 270.489,A -85,B 0,C 180,E1 -5983.235,E2 -5983.235} C_VEL
LIN {X 0,Y 502.74,Z 270.485,A -85,B 0,C 180,E1 -5985.655,E2 -5985.655} C_VEL
LIN {X 0,Y 502.75,Z 270.486,A -85,B 0,C 180,E1 -5989.014,E2 -5989.014} C_VEL
LIN {X 0,Y 502.745,Z 270.481,A -85,B 0,C 180,E1 -5992.041,E2 -5992.041} C_VEL
LIN {X 0,Y 502.77,Z 270.486,A -85,B 0,C 180,E1 -5995.031,E2 -5995.031} C_VEL
LIN {X 0,Y 502.759,Z 270.483,A -85,B 0,C 180,E1 -5997.177,E2 -5997.177} C_VEL
LIN {X 0,Y 502.07,Z 270.567,A -85,B 0,C 180,E1 -5997.845,E2 -5997.845} C_VEL
LIN {X 0,Y 499.2,Z 270.927,A -85,B 0,C 180,E1 -5998.931,E2 -5998.931} C_VEL
LIN {X 0,Y 496.79,Z 271.226,A -85,B 0,C 180,E1 -5999.806,E2 -5999.806} C_VEL
LIN {X 0,Y 495.762,Z 271.355,A -85,B 0,C 180,E1 -6000.482,E2 -6000.482} C_VEL
LIN {X 0,Y 495.681,Z 271.364,A -85,B 0,C 180,E1 -6000.711,E2 -6000.711} C_VEL
LIN {X 0,Y 495.722,Z 271.363,A -85,B 0,C 180,E1 -6003.274,E2 -6003.274} C_VEL
LIN {X 0,Y 495.739,Z 271.436,A -85,B 0,C 180,E1 -6004.801,E2 -6004.801} C_VEL
LIN {X 0,Y 498.301,Z 283.285,A -85,B 0,C 180,E1 -6006.959,E2 -6006.959} C_VEL
LIN {X 0,Y 498.425,Z 285.447,A -85,B 0,C 180,E1 -6007.323,E2 -6007.323} C_VEL
LIN {X 0,Y 502.213,Z 301.378,A -85,B 0,C 180,E1 -6007.748,E2 -6007.748} C_VEL
LIN {X 0,Y 501.227,Z 415.469,A -85,B 0,C 180,E1 -6009.426,E2 -6009.426} C_VEL
LIN {X 0,Y 500.895,Z 451.533,A -85,B 0,C 180,E1 -6009.985,E2 -6009.985} C_VEL
LIN {X 0,Y 500.591,Z 466.113,A -85,B 0,C 180,E1 -6010.364,E2 -6010.364} C_VEL
LIN {X 0,Y 500.098,Z 481.292,A -85,B 0,C 180,E1 -6010.93,E2 -6010.93} C_VEL
LIN {X 0,Y 499.518,Z 495.836,A -85,B 0,C 180,E1 -6011.65,E2 -6011.65} C_VEL
LIN {X 0,Y 498.883,Z 509.085,A -85,B 0,C 180,E1 -6012.475,E2 -6012.475} C_VEL
LIN {X 0,Y 498.217,Z 522.545,A -85,B 0,C 180,E1 -6013.507,E2 -6013.507} C_VEL
LIN {X 0,Y 497.546,Z 534.745,A -85,B 0,C 180,E1 -6014.642,E2 -6014.642} C_VEL
LIN {X 0,Y 496.935,Z 545.85,A -85,B 0,C 180,E1 -6015.879,E2 -6015.879} C_VEL
LIN {X 0,Y 496.359,Z 556.636,A -85,B 0,C 180,E1 -6017.322,E2 -6017.322} C_VEL
LIN {X 0,Y 495.965,Z 565.578,A -85,B 0,C 180,E1 -6018.764,E2 -6018.764} C_VEL
LIN {X 0,Y 495.622,Z 572.989,A -85,B 0,C 180,E1 -6020.202,E2 -6020.202} C_VEL
LIN {X 0,Y 495.352,Z 579.916,A -85,B 0,C 180,E1 -6021.843,E2 -6021.843} C_VEL
LIN {X 0,Y 495.164,Z 585.361,A -85,B 0,C 180,E1 -6023.48,E2 -6023.48} C_VEL
LIN {X 0,Y 495.198,Z 587.571,A -85,B 0,C 180,E1 -6024.298,E2 -6024.298} C_VEL
LIN {X 0,Y 495.093,Z 591.062,A -85,B 0,C 180,E1 -6025.93,E2 -6025.93} C_VEL
LIN {X 0,Y 495.05,Z 593.372,A -85,B 0,C 180,E1 -6027.559,E2 -6027.559} C_VEL
LIN {X 0,Y 494.907,Z 594.56,A -85,B 0,C 180,E1 -6029.186,E2 -6029.186} C_VEL
LIN {X 0,Y 494.908,Z 594.578,A -85,B 0,C 180,E1 -6030.813,E2 -6030.813} C_VEL
LIN {X 0,Y 495.051,Z 593.464,A -85,B 0,C 180,E1 -6032.441,E2 -6032.441} C_VEL
LIN {X 0,Y 495.093,Z 591.226,A -85,B 0,C 180,E1 -6034.07,E2 -6034.07} C_VEL
LIN {X 0,Y 495.187,Z 587.804,A -85,B 0,C 180,E1 -6035.701,E2 -6035.701} C_VEL
LIN {X 0,Y 495.245,Z 583.122,A -85,B 0,C 180,E1 -6037.337,E2 -6037.337} C_VEL
LIN {X 0,Y 495.453,Z 577.049,A -85,B 0,C 180,E1 -6038.976,E2 -6038.976} C_VEL
LIN {X 0,Y 495.748,Z 569.399,A -85,B 0,C 180,E1 -6040.62,E2 -6040.62} C_VEL
LIN {X 0,Y 496.15,Z 560.297,A -85,B 0,C 180,E1 -6042.207,E2 -6042.207} C_VEL
LIN {X 0,Y 496.658,Z 551.404,A -85,B 0,C 180,E1 -6043.502,E2 -6043.502} C_VEL
LIN {X 0,Y 497.21,Z 541.315,A -85,B 0,C 180,E1 -6044.739,E2 -6044.739} C_VEL
LIN {X 0,Y 497.766,Z 530.249,A -85,B 0,C 180,E1 -6045.887,E2 -6045.887} C_VEL
LIN {X 0,Y 498.425,Z 518.535,A -85,B 0,C 180,E1 -6046.907,E2 -6046.907} C_VEL
LIN {X 0,Y 499.088,Z 505.729,A -85,B 0,C 180,E1 -6047.835,E2 -6047.835} C_VEL
LIN {X 0,Y 499.67,Z 491.681,A -85,B 0,C 180,E1 -6048.662,E2 -6048.662} C_VEL
LIN {X 0,Y 500.237,Z 477.459,A -85,B 0,C 180,E1 -6049.316,E2 -6049.316} C_VEL
LIN {X 0,Y 500.61,Z 462.58,A -85,B 0,C 180,E1 -6049.831,E2 -6049.831} C_VEL
LIN {X 0,Y 500.962,Z 447.454,A -85,B 0,C 180,E1 -6050.183,E2 -6050.183} C_VEL
LIN {X 0,Y 502.174,Z 314.31,A -85,B 0,C 180,E1 -6052.148,E2 -6052.148} C_VEL
LIN {X 0,Y 502.076,Z 300.717,A -85,B 0,C 180,E1 -6052.359,E2 -6052.359} C_VEL
LIN {X 0,Y 498.473,Z 285.385,A -85,B 0,C 180,E1 -6052.775,E2 -6052.775} C_VEL
LIN {X 0,Y 497.642,Z 279.851,A -85,B 0,C 180,E1 -6053.745,E2 -6053.745} C_VEL
LIN {X 0,Y 495.73,Z 271.363,A -85,B 0,C 180,E1 -6055.338,E2 -6055.338} C_VEL
LIN {X 0,Y 495.732,Z 271.361,A -85,B 0,C 180,E1 -6058.481,E2 -6058.481} C_VEL
LIN {X 0,Y 495.728,Z 271.362,A -85,B 0,C 180,E1 -6061.638,E2 -6061.638} C_VEL
LIN {X 0,Y 495.751,Z 271.362,A -85,B 0,C 180,E1 -6064.691,E2 -6064.691} C_VEL
LIN {X 0,Y 495.699,Z 271.363,A -85,B 0,C 180,E1 -6067.564,E2 -6067.564} C_VEL
LIN {X 0,Y 495.741,Z 271.355,A -85,B 0,C 180,E1 -6070.044,E2 -6070.044} C_VEL
LIN {X 0,Y 495.687,Z 271.361,A -85,B 0,C 180,E1 -6072.887,E2 -6072.887} C_VEL
LIN {X 0,Y 495.71,Z 271.359,A -85,B 0,C 180,E1 -6075.996,E2 -6075.996} C_VEL
LIN {X 0,Y 495.706,Z 271.36,A -85,B 0,C 180,E1 -6079.294,E2 -6079.294} C_VEL
LIN {X 0,Y 495.706,Z 271.358,A -85,B 0,C 180,E1 -6081.404,E2 -6081.404} C_VEL
LIN {X 0,Y 495.716,Z 271.351,A -85,B 0,C 180,E1 -6084.459,E2 -6084.459} C_VEL
LIN {X 0,Y 495.722,Z 271.357,A -85,B 0,C 180,E1 -6087.402,E2 -6087.402} C_VEL
LIN {X 0,Y 495.693,Z 271.363,A -85,B 0,C 180,E1 -6090.249,E2 -6090.249} C_VEL
LIN {X 0,Y 495.735,Z 271.355,A -85,B 0,C 180,E1 -6093.271,E2 -6093.271} C_VEL
LIN {X 0,Y 495.728,Z 271.359,A -85,B 0,C 180,E1 -6096.612,E2 -6096.612} C_VEL
LIN {X 0,Y 495.765,Z 271.351,A -85,B 0,C 180,E1 -6099.328,E2 -6099.328} C_VEL
LIN {X 0,Y 495.759,Z 271.349,A -85,B 0,C 180,E1 -6101.827,E2 -6101.827} C_VEL
LIN {X 0,Y 495.772,Z 271.347,A -85,B 0,C 180,E1 -6105.217,E2 -6105.217} C_VEL
LIN {X 0,Y 495.848,Z 271.346,A -85,B 0,C 180,E1 -6108.555,E2 -6108.555} C_VEL
LIN {X 0,Y 495.811,Z 271.344,A -85,B 0,C 180,E1 -6111.851,E2 -6111.851} C_VEL
LIN {X 0,Y 495.816,Z 271.342,A -85,B 0,C 180,E1 -6115.121,E2 -6115.121} C_VEL
LIN {X 0,Y 495.981,Z 271.324,A -85,B 0,C 180,E1 -6117.564,E2 -6117.564} C_VEL
LIN {X 0,Y 495.94,Z 271.326,A -85,B 0,C 180,E1 -6120.812,E2 -6120.812} C_VEL
LIN {X 0,Y 495.98,Z 271.329,A -85,B 0,C 180,E1 -6122.436,E2 -6122.436} C_VEL
LIN {X 0,Y 495.869,Z 271.339,A -85,B 0,C 180,E1 -6125.694,E2 -6125.694} C_VEL
LIN {X 0,Y 495.829,Z 271.343,A -85,B 0,C 180,E1 -6128.97,E2 -6128.97} C_VEL
LIN {X 0,Y 495.827,Z 271.349,A -85,B 0,C 180,E1 -6132.035,E2 -6132.035} C_VEL
LIN {X 0,Y 495.823,Z 271.342,A -85,B 0,C 180,E1 -6135.451,E2 -6135.451} C_VEL
LIN {X 0,Y 495.777,Z 271.348,A -85,B 0,C 180,E1 -6139.029,E2 -6139.029} C_VEL
LIN {X 0,Y 495.741,Z 271.359,A -85,B 0,C 180,E1 -6141.629,E2 -6141.629} C_VEL
LIN {X 0,Y 495.721,Z 271.349,A -85,B 0,C 180,E1 -6144.277,E2 -6144.277} C_VEL
LIN {X 0,Y 495.758,Z 271.348,A -85,B 0,C 180,E1 -6146.977,E2 -6146.977} C_VEL
LIN {X 0,Y 495.763,Z 271.351,A -85,B 0,C 180,E1 -6150.147,E2 -6150.147} C_VEL
LIN {X 0,Y 495.792,Z 271.344,A -85,B 0,C 180,E1 -6153.244,E2 -6153.244} C_VEL
LIN {X 0,Y 495.72,Z 271.356,A -85,B 0,C 180,E1 -6156.089,E2 -6156.089} C_VEL
LIN {X 0,Y 495.761,Z 271.35,A -85,B 0,C 180,E1 -6158.768,E2 -6158.768} C_VEL
LIN {X 0,Y 495.754,Z 271.36,A -85,B 0,C 180,E1 -6161.781,E2 -6161.781} C_VEL
LIN {X 0,Y 495.735,Z 271.357,A -85,B 0,C 180,E1 -6165.141,E2 -6165.141} C_VEL
LIN {X 0,Y 495.754,Z 271.352,A -85,B 0,C 180,E1 -6168.219,E2 -6168.219} C_VEL
LIN {X 0,Y 495.749,Z 271.359,A -85,B 0,C 180,E1 -6171.409,E2 -6171.409} C_VEL
LIN {X 0,Y 495.754,Z 271.355,A -85,B 0,C 180,E1 -6174.463,E2 -6174.463} C_VEL
LIN {X 0,Y 495.766,Z 271.357,A -85,B 0,C 180,E1 -6177.406,E2 -6177.406} C_VEL
LIN {X 0,Y 495.831,Z 271.517,A -85,B 0,C 180,E1 -6180.434,E2 -6180.434} C_VEL
LIN {X 0,Y 499.528,Z 287.275,A -85,B 0,C 180,E1 -6182.881,E2 -6182.881} C_VEL
LIN {X 0,Y 499.396,Z 294.719,A -85,B 0,C 180,E1 -6183.91,E2 -6183.91} C_VEL
LIN {X 0,Y 498.643,Z 312.814,A -85,B 0,C 180,E1 -6186.366,E2 -6186.366} C_VEL
LIN {X 0,Y 498.316,Z 319.351,A -85,B 0,C 180,E1 -6187.247,E2 -6187.247} C_VEL
LIN {X 0,Y 502.095,Z 339.995,A -85,B 0,C 180,E1 -6187.746,E2 -6187.746} C_VEL
LIN {X 0,Y 500.762,Z 485.967,A -85,B 0,C 180,E1 -6189.902,E2 -6189.902} C_VEL
LIN {X 0,Y 500.396,Z 500.855,A -85,B 0,C 180,E1 -6190.275,E2 -6190.275} C_VEL
LIN {X 0,Y 499.882,Z 515.351,A -85,B 0,C 180,E1 -6190.794,E2 -6190.794} C_VEL
LIN {X 0,Y 499.267,Z 528.894,A -85,B 0,C 180,E1 -6191.429,E2 -6191.429} C_VEL
LIN {X 0,Y 498.682,Z 542.834,A -85,B 0,C 180,E1 -6192.256,E2 -6192.256} C_VEL
LIN {X 0,Y 497.99,Z 555.605,A -85,B 0,C 180,E1 -6193.184,E2 -6193.184} C_VEL
LIN {X 0,Y 497.358,Z 568.306,A -85,B 0,C 180,E1 -6194.3,E2 -6194.3} C_VEL
LIN {X 0,Y 496.756,Z 579.352,A -85,B 0,C 180,E1 -6195.456,E2 -6195.456} C_VEL
LIN {X 0,Y 496.292,Z 589.373,A -85,B 0,C 180,E1 -6196.696,E2 -6196.696} C_VEL
LIN {X 0,Y 495.815,Z 599.056,A -85,B 0,C 180,E1 -6198.119,E2 -6198.119} C_VEL
LIN {X 0,Y 495.557,Z 607.366,A -85,B 0,C 180,E1 -6199.583,E2 -6199.583} C_VEL
LIN {X 0,Y 495.284,Z 614.132,A -85,B 0,C 180,E1 -6201.02,E2 -6201.02} C_VEL
LIN {X 0,Y 495.159,Z 620.387,A -85,B 0,C 180,E1 -6202.661,E2 -6202.661} C_VEL
LIN {X 0,Y 495.068,Z 625.225,A -85,B 0,C 180,E1 -6204.297,E2 -6204.297} C_VEL
LIN {X 0,Y 494.993,Z 628.769,A -85,B 0,C 180,E1 -6205.929,E2 -6205.929} C_VEL
LIN {X 0,Y 494.994,Z 631.102,A -85,B 0,C 180,E1 -6207.559,E2 -6207.559} C_VEL
LIN {X 0,Y 494.908,Z 632.272,A -85,B 0,C 180,E1 -6209.187,E2 -6209.187} C_VEL
LIN {X 0,Y 494.908,Z 632.271,A -85,B 0,C 180,E1 -6210.814,E2 -6210.814} C_VEL
LIN {X 0,Y 494.994,Z 631.097,A -85,B 0,C 180,E1 -6212.442,E2 -6212.442} C_VEL
LIN {X 0,Y 494.993,Z 628.763,A -85,B 0,C 180,E1 -6214.071,E2 -6214.071} C_VEL
LIN {X 0,Y 495.064,Z 625.224,A -85,B 0,C 180,E1 -6215.703,E2 -6215.703} C_VEL
LIN {X 0,Y 495.16,Z 620.388,A -85,B 0,C 180,E1 -6217.339,E2 -6217.339} C_VEL
LIN {X 0,Y 495.285,Z 614.125,A -85,B 0,C 180,E1 -6218.98,E2 -6218.98} C_VEL
LIN {X 0,Y 495.605,Z 606.266,A -85,B 0,C 180,E1 -6220.624,E2 -6220.624} C_VEL
LIN {X 0,Y 495.87,Z 597.973,A -85,B 0,C 180,E1 -6222.057,E2 -6222.057} C_VEL
LIN {X 0,Y 496.374,Z 587.843,A -85,B 0,C 180,E1 -6223.511,E2 -6223.511} C_VEL
LIN {X 0,Y 496.827,Z 577.55,A -85,B 0,C 180,E1 -6224.752,E2 -6224.752} C_VEL
LIN {X 0,Y 497.515,Z 565.099,A -85,B 0,C 180,E1 -6226.009,E2 -6226.009} C_VEL
LIN {X 0,Y 498.173,Z 551.666,A -85,B 0,C 180,E1 -6227.128,E2 -6227.128} C_VEL
LIN {X 0,Y 498.94,Z 538.008,A -85,B 0,C 180,E1 -6228.053,E2 -6228.053} C_VEL
LIN {X 0,Y 499.518,Z 523.864,A -85,B 0,C 180,E1 -6228.828,E2 -6228.828} C_VEL
LIN {X 0,Y 500.128,Z 508.67,A -85,B 0,C 180,E1 -6229.467,E2 -6229.467} C_VEL
LIN {X 0,Y 500.59,Z 493.416,A -85,B 0,C 180,E1 -6229.932,E2 -6229.932} C_VEL
LIN {X 0,Y 500.858,Z 477.501,A -85,B 0,C 180,E1 -6230.242,E2 -6230.242} C_VEL
LIN {X 0,Y 502.084,Z 339.922,A -85,B 0,C 180,E1 -6232.255,E2 -6232.255} C_VEL
LIN {X 0,Y 498.342,Z 319.214,A -85,B 0,C 180,E1 -6232.77,E2 -6232.77} C_VEL
LIN {X 0,Y 499.203,Z 300.107,A -85,B 0,C 180,E1 -6235.353,E2 -6235.353} C_VEL
LIN {X 0,Y 499.679,Z 288.559,A -85,B 0,C 180,E1 -6236.93,E2 -6236.93} C_VEL
LIN {X 0,Y 498.265,Z 281.702,A -85,B 0,C 180,E1 -6237.969,E2 -6237.969} C_VEL
LIN {X 0,Y 495.815,Z 271.349,A -85,B 0,C 180,E1 -6239.627,E2 -6239.627} C_VEL
LIN {X 0,Y 495.795,Z 271.351,A -85,B 0,C 180,E1 -6243.245,E2 -6243.245} C_VEL
LIN {X 0,Y 495.722,Z 271.361,A -85,B 0,C 180,E1 -6246.089,E2 -6246.089} C_VEL
LIN {X 0,Y 495.766,Z 271.352,A -85,B 0,C 180,E1 -6248.769,E2 -6248.769} C_VEL
LIN {X 0,Y 495.753,Z 271.354,A -85,B 0,C 180,E1 -6251.782,E2 -6251.782} C_VEL
LIN {X 0,Y 495.74,Z 271.355,A -85,B 0,C 180,E1 -6255.141,E2 -6255.141} C_VEL
LIN {X 0,Y 495.759,Z 271.357,A -85,B 0,C 180,E1 -6258.219,E2 -6258.219} C_VEL
LIN {X 0,Y 495.75,Z 271.353,A -85,B 0,C 180,E1 -6261.408,E2 -6261.408} C_VEL
LIN {X 0,Y 495.748,Z 271.357,A -85,B 0,C 180,E1 -6264.462,E2 -6264.462} C_VEL
LIN {X 0,Y 495.772,Z 271.348,A -85,B 0,C 180,E1 -6267.406,E2 -6267.406} C_VEL
LIN {X 0,Y 495.767,Z 271.354,A -85,B 0,C 180,E1 -6270.254,E2 -6270.254} C_VEL
LIN {X 0,Y 495.764,Z 271.349,A -85,B 0,C 180,E1 -6273.266,E2 -6273.266} C_VEL
LIN {X 0,Y 495.746,Z 271.352,A -85,B 0,C 180,E1 -6276.613,E2 -6276.613} C_VEL
LIN {X 0,Y 495.784,Z 271.349,A -85,B 0,C 180,E1 -6279.324,E2 -6279.324} C_VEL
LIN {X 0,Y 495.784,Z 271.351,A -85,B 0,C 180,E1 -6281.829,E2 -6281.829} C_VEL
LIN {X 0,Y 495.794,Z 271.345,A -85,B 0,C 180,E1 -6285.217,E2 -6285.217} C_VEL
LIN {X 0,Y 495.856,Z 271.338,A -85,B 0,C 180,E1 -6288.555,E2 -6288.555} C_VEL
LIN {X 0,Y 495.819,Z 271.351,A -85,B 0,C 180,E1 -6291.851,E2 -6291.851} C_VEL
LIN {X 0,Y 495.861,Z 271.343,A -85,B 0,C 180,E1 -6294.306,E2 -6294.306} C_VEL
LIN {X 0,Y 495.981,Z 271.326,A -85,B 0,C 180,E1 -6297.564,E2 -6297.564} C_VEL
LIN {X 0,Y 495.976,Z 271.33,A -85,B 0,C 180,E1 -6300,E2 -6300} C_VEL
LIN {X 0,Y 495.987,Z 271.324,A -85,B 0,C 180,E1 -6302.436,E2 -6302.436} C_VEL
LIN {X 0,Y 495.85,Z 271.345,A -85,B 0,C 180,E1 -6305.694,E2 -6305.694} C_VEL
LIN {X 0,Y 495.817,Z 271.348,A -85,B 0,C 180,E1 -6308.149,E2 -6308.149} C_VEL
LIN {X 0,Y 495.854,Z 271.342,A -85,B 0,C 180,E1 -6311.445,E2 -6311.445} C_VEL
LIN {X 0,Y 495.778,Z 271.346,A -85,B 0,C 180,E1 -6314.783,E2 -6314.783} C_VEL
LIN {X 0,Y 495.752,Z 271.351,A -85,B 0,C 180,E1 -6318.226,E2 -6318.226} C_VEL
LIN {X 0,Y 495.75,Z 271.353,A -85,B 0,C 180,E1 -6320.758,E2 -6320.758} C_VEL
LIN {X 0,Y 495.734,Z 271.358,A -85,B 0,C 180,E1 -6323.388,E2 -6323.388} C_VEL
LIN {X 0,Y 495.711,Z 271.356,A -85,B 0,C 180,E1 -6326.072,E2 -6326.072} C_VEL
LIN {X 0,Y 495.699,Z 271.351,A -85,B 0,C 180,E1 -6328.82,E2 -6328.82} C_VEL
LIN {X 0,Y 495.733,Z 271.359,A -85,B 0,C 180,E1 -6331.72,E2 -6331.72} C_VEL
LIN {X 0,Y 495.741,Z 271.355,A -85,B 0,C 180,E1 -6334.688,E2 -6334.688} C_VEL
LIN {X 0,Y 495.694,Z 271.365,A -85,B 0,C 180,E1 -6337.565,E2 -6337.565} C_VEL
LIN {X 0,Y 495.708,Z 271.358,A -85,B 0,C 180,E1 -6340.039,E2 -6340.039} C_VEL
LIN {X 0,Y 495.692,Z 271.363,A -85,B 0,C 180,E1 -6342.887,E2 -6342.887} C_VEL
LIN {X 0,Y 495.713,Z 271.364,A -85,B 0,C 180,E1 -6345.144,E2 -6345.144} C_VEL
LIN {X 0,Y 495.7,Z 271.358,A -85,B 0,C 180,E1 -6348.212,E2 -6348.212} C_VEL
LIN {X 0,Y 495.708,Z 271.363,A -85,B 0,C 180,E1 -6351.404,E2 -6351.404} C_VEL
LIN {X 0,Y 495.72,Z 271.359,A -85,B 0,C 180,E1 -6354.459,E2 -6354.459} C_VEL
LIN {X 0,Y 495.726,Z 271.361,A -85,B 0,C 180,E1 -6357.402,E2 -6357.402} C_VEL
LIN {X 0,Y 495.697,Z 271.362,A -85,B 0,C 180,E1 -6360.249,E2 -6360.249} C_VEL
LIN {X 0,Y 495.681,Z 271.364,A -85,B 0,C 180,E1 -6360.711,E2 -6360.711} C_VEL
LIN {X 0,Y 495.016,Z 271.451,A -85,B 0,C 180,E1 -6361.39,E2 -6361.39} C_VEL
LIN {X 0,Y 492.153,Z 271.804,A -85,B 0,C 180,E1 -6362.492,E2 -6362.492} C_VEL
LIN {X 0,Y 489.75,Z 272.106,A -85,B 0,C 180,E1 -6363.381,E2 -6363.381} C_VEL
LIN {X 0,Y 488.749,Z 272.229,A -85,B 0,C 180,E1 -6364.067,E2 -6364.067} C_VEL
LIN {X 0,Y 488.683,Z 272.238,A -85,B 0,C 180,E1 -6364.299,E2 -6364.299} C_VEL
LIN {X 0,Y 488.675,Z 272.244,A -85,B 0,C 180,E1 -6364.51,E2 -6364.51} C_VEL
LIN {X 0,Y 491.444,Z 284.874,A -85,B 0,C 180,E1 -6366.841,E2 -6366.841} C_VEL
LIN {X 0,Y 491.572,Z 285.806,A -85,B 0,C 180,E1 -6366.99,E2 -6366.99} C_VEL
LIN {X 0,Y 495.71,Z 303.098,A -85,B 0,C 180,E1 -6367.462,E2 -6367.462} C_VEL
LIN {X 0,Y 494.316,Z 447.885,A -85,B 0,C 180,E1 -6369.628,E2 -6369.628} C_VEL
LIN {X 0,Y 493.986,Z 462.96,A -85,B 0,C 180,E1 -6369.985,E2 -6369.985} C_VEL
LIN {X 0,Y 493.515,Z 478.049,A -85,B 0,C 180,E1 -6370.514,E2 -6370.514} C_VEL
LIN {X 0,Y 492.907,Z 492.244,A -85,B 0,C 180,E1 -6371.18,E2 -6371.18} C_VEL
LIN {X 0,Y 492.317,Z 506.226,A -85,B 0,C 180,E1 -6372.018,E2 -6372.018} C_VEL
LIN {X 0,Y 491.594,Z 519,A -85,B 0,C 180,E1 -6372.957,E2 -6372.957} C_VEL
LIN {X 0,Y 490.927,Z 531.319,A -85,B 0,C 180,E1 -6374.056,E2 -6374.056} C_VEL
LIN {X 0,Y 490.242,Z 542.594,A -85,B 0,C 180,E1 -6375.258,E2 -6375.258} C_VEL
LIN {X 0,Y 489.653,Z 552.518,A -85,B 0,C 180,E1 -6376.512,E2 -6376.512} C_VEL
LIN {X 0,Y 489.131,Z 561.527,A -85,B 0,C 180,E1 -6377.858,E2 -6377.858} C_VEL
LIN {X 0,Y 488.709,Z 570.271,A -85,B 0,C 180,E1 -6379.434,E2 -6379.434} C_VEL
LIN {X 0,Y 488.434,Z 576.924,A -85,B 0,C 180,E1 -6380.893,E2 -6380.893} C_VEL
LIN {X 0,Y 488.193,Z 583.087,A -85,B 0,C 180,E1 -6382.555,E2 -6382.555} C_VEL
LIN {X 0,Y 488.134,Z 587.843,A -85,B 0,C 180,E1 -6384.215,E2 -6384.215} C_VEL
LIN {X 0,Y 487.995,Z 591.334,A -85,B 0,C 180,E1 -6385.87,E2 -6385.87} C_VEL
LIN {X 0,Y 487.956,Z 593.643,A -85,B 0,C 180,E1 -6387.523,E2 -6387.523} C_VEL
LIN {X 0,Y 487.831,Z 594.829,A -85,B 0,C 180,E1 -6389.174,E2 -6389.174} C_VEL
LIN {X 0,Y 487.831,Z 594.848,A -85,B 0,C 180,E1 -6390.825,E2 -6390.825} C_VEL
LIN {X 0,Y 487.956,Z 593.734,A -85,B 0,C 180,E1 -6392.476,E2 -6392.476} C_VEL
LIN {X 0,Y 487.995,Z 591.496,A -85,B 0,C 180,E1 -6394.129,E2 -6394.129} C_VEL
LIN {X 0,Y 488.124,Z 588.073,A -85,B 0,C 180,E1 -6395.784,E2 -6395.784} C_VEL
LIN {X 0,Y 488.191,Z 583.391,A -85,B 0,C 180,E1 -6397.444,E2 -6397.444} C_VEL
LIN {X 0,Y 488.426,Z 577.317,A -85,B 0,C 180,E1 -6399.107,E2 -6399.107} C_VEL
LIN {X 0,Y 488.757,Z 569.667,A -85,B 0,C 180,E1 -6400.773,E2 -6400.773} C_VEL
LIN {X 0,Y 489.16,Z 561.007,A -85,B 0,C 180,E1 -6402.315,E2 -6402.315} C_VEL
LIN {X 0,Y 489.749,Z 551.669,A -85,B 0,C 180,E1 -6403.696,E2 -6403.696} C_VEL
LIN {X 0,Y 490.327,Z 541.581,A -85,B 0,C 180,E1 -6404.951,E2 -6404.951} C_VEL
LIN {X 0,Y 490.918,Z 530.782,A -85,B 0,C 180,E1 -6406.088,E2 -6406.088} C_VEL
LIN {X 0,Y 491.631,Z 518.799,A -85,B 0,C 180,E1 -6407.148,E2 -6407.148} C_VEL
LIN {X 0,Y 492.325,Z 505.991,A -85,B 0,C 180,E1 -6408.088,E2 -6408.088} C_VEL
LIN {X 0,Y 492.939,Z 491.942,A -85,B 0,C 180,E1 -6408.926,E2 -6408.926} C_VEL
LIN {X 0,Y 493.574,Z 476.935,A -85,B 0,C 180,E1 -6409.62,E2 -6409.62} C_VEL
LIN {X 0,Y 493.969,Z 462.013,A -85,B 0,C 180,E1 -6410.133,E2 -6410.133} C_VEL
LIN {X 0,Y 494.308,Z 447.695,A -85,B 0,C 180,E1 -6410.466,E2 -6410.466} C_VEL
LIN {X 0,Y 495.52,Z 323.392,A -85,B 0,C 180,E1 -6412.325,E2 -6412.325} C_VEL
LIN {X 0,Y 495.663,Z 302.449,A -85,B 0,C 180,E1 -6412.641,E2 -6412.641} C_VEL
LIN {X 0,Y 491.578,Z 285.642,A -85,B 0,C 180,E1 -6413.115,E2 -6413.115} C_VEL
LIN {X 0,Y 488.713,Z 272.235,A -85,B 0,C 180,E1 -6415.614,E2 -6415.614} C_VEL
LIN {X 0,Y 488.677,Z 272.241,A -85,B 0,C 180,E1 -6418.683,E2 -6418.683} C_VEL
LIN {X 0,Y 488.665,Z 272.243,A -85,B 0,C 180,E1 -6421.181,E2 -6421.181} C_VEL
LIN {X 0,Y 488.707,Z 272.234,A -85,B 0,C 180,E1 -6424.114,E2 -6424.114} C_VEL
LIN {X 0,Y 488.649,Z 272.245,A -85,B 0,C 180,E1 -6427.161,E2 -6427.161} C_VEL
LIN {X 0,Y 488.692,Z 272.235,A -85,B 0,C 180,E1 -6430.341,E2 -6430.341} C_VEL
LIN {X 0,Y 488.662,Z 272.233,A -85,B 0,C 180,E1 -6433.657,E2 -6433.657} C_VEL
LIN {X 0,Y 488.662,Z 272.239,A -85,B 0,C 180,E1 -6436.343,E2 -6436.343} C_VEL
LIN {X 0,Y 488.665,Z 272.235,A -85,B 0,C 180,E1 -6439.67,E2 -6439.67} C_VEL
LIN {X 0,Y 488.638,Z 272.233,A -85,B 0,C 180,E1 -6442.837,E2 -6442.837} C_VEL
LIN {X 0,Y 488.701,Z 272.23,A -85,B 0,C 180,E1 -6445.885,E2 -6445.885} C_VEL
LIN {X 0,Y 488.656,Z 272.241,A -85,B 0,C 180,E1 -6448.818,E2 -6448.818} C_VEL
LIN {X 0,Y 488.682,Z 272.233,A -85,B 0,C 180,E1 -6451.667,E2 -6451.667} C_VEL
LIN {X 0,Y 488.656,Z 272.243,A -85,B 0,C 180,E1 -6454.439,E2 -6454.439} C_VEL
LIN {X 0,Y 488.704,Z 272.23,A -85,B 0,C 180,E1 -6457.152,E2 -6457.152} C_VEL
LIN {X 0,Y 488.692,Z 272.233,A -85,B 0,C 180,E1 -6459.809,E2 -6459.809} C_VEL
LIN {X 0,Y 488.667,Z 272.24,A -85,B 0,C 180,E1 -6462.421,E2 -6462.421} C_VEL
LIN {X 0,Y 488.744,Z 272.224,A -85,B 0,C 180,E1 -6464.999,E2 -6464.999} C_VEL
LIN {X 0,Y 488.803,Z 272.226,A -85,B 0,C 180,E1 -6468.387,E2 -6468.387} C_VEL
LIN {X 0,Y 488.758,Z 272.222,A -85,B 0,C 180,E1 -6471.733,E2 -6471.733} C_VEL
LIN {X 0,Y 488.804,Z 272.225,A -85,B 0,C 180,E1 -6474.224,E2 -6474.224} C_VEL
LIN {X 0,Y 488.948,Z 272.2,A -85,B 0,C 180,E1 -6477.528,E2 -6477.528} C_VEL
LIN {X 0,Y 488.892,Z 272.203,A -85,B 0,C 180,E1 -6480.824,E2 -6480.824} C_VEL
LIN {X 0,Y 488.947,Z 272.205,A -85,B 0,C 180,E1 -6482.471,E2 -6482.471} C_VEL
LIN {X 0,Y 488.826,Z 272.217,A -85,B 0,C 180,E1 -6485.776,E2 -6485.776} C_VEL
LIN {X 0,Y 488.768,Z 272.229,A -85,B 0,C 180,E1 -6488.267,E2 -6488.267} C_VEL
LIN {X 0,Y 488.804,Z 272.217,A -85,B 0,C 180,E1 -6491.612,E2 -6491.612} C_VEL
LIN {X 0,Y 488.76,Z 272.22,A -85,B 0,C 180,E1 -6495,E2 -6495} C_VEL
LIN {X 0,Y 488.744,Z 272.226,A -85,B 0,C 180,E1 -6498.442,E2 -6498.442} C_VEL
LIN {X 0,Y 488.706,Z 272.231,A -85,B 0,C 180,E1 -6501.071,E2 -6501.071} C_VEL
LIN {X 0,Y 488.674,Z 272.235,A -85,B 0,C 180,E1 -6503.746,E2 -6503.746} C_VEL
LIN {X 0,Y 488.717,Z 272.227,A -85,B 0,C 180,E1 -6506.474,E2 -6506.474} C_VEL
LIN {X 0,Y 488.709,Z 272.232,A -85,B 0,C 180,E1 -6509.271,E2 -6509.271} C_VEL
LIN {X 0,Y 488.702,Z 272.227,A -85,B 0,C 180,E1 -6512.147,E2 -6512.147} C_VEL
LIN {X 0,Y 488.717,Z 272.231,A -85,B 0,C 180,E1 -6515.115,E2 -6515.115} C_VEL
LIN {X 0,Y 488.678,Z 272.234,A -85,B 0,C 180,E1 -6518.2,E2 -6518.2} C_VEL
LIN {X 0,Y 488.717,Z 272.23,A -85,B 0,C 180,E1 -6520.345,E2 -6520.345} C_VEL
LIN {X 0,Y 488.682,Z 272.24,A -85,B 0,C 180,E1 -6523.655,E2 -6523.655} C_VEL
LIN {X 0,Y 488.682,Z 272.233,A -85,B 0,C 180,E1 -6526.345,E2 -6526.345} C_VEL
LIN {X 0,Y 488.731,Z 272.23,A -85,B 0,C 180,E1 -6529.677,E2 -6529.677} C_VEL
LIN {X 0,Y 488.68,Z 272.235,A -85,B 0,C 180,E1 -6532.842,E2 -6532.842} C_VEL
LIN {X 0,Y 488.733,Z 272.23,A -85,B 0,C 180,E1 -6535.888,E2 -6535.888} C_VEL
LIN {X 0,Y 488.691,Z 272.238,A -85,B 0,C 180,E1 -6538.821,E2 -6538.821} C_VEL
LIN {X 0,Y 488.755,Z 272.265,A -85,B 0,C 180,E1 -6540.11,E2 -6540.11} C_VEL
LIN {X 0,Y 492.615,Z 288.476,A -85,B 0,C 180,E1 -6542.676,E2 -6542.676} C_VEL
LIN {X 0,Y 492.728,Z 292.847,A -85,B 0,C 180,E1 -6543.302,E2 -6543.302} C_VEL
LIN {X 0,Y 491.898,Z 311.748,A -85,B 0,C 180,E1 -6545.91,E2 -6545.91} C_VEL
LIN {X 0,Y 491.514,Z 319.077,A -85,B 0,C 180,E1 -6546.914,E2 -6546.914} C_VEL
LIN {X 0,Y 495.519,Z 340.865,A -85,B 0,C 180,E1 -6547.452,E2 -6547.452} C_VEL
LIN {X 0,Y 494.122,Z 485.006,A -85,B 0,C 180,E1 -6549.607,E2 -6549.607} C_VEL
LIN {X 0,Y 493.672,Z 500.675,A -85,B 0,C 180,E1 -6549.997,E2 -6549.997} C_VEL
LIN {X 0,Y 493.104,Z 516.687,A -85,B 0,C 180,E1 -6550.588,E2 -6550.588} C_VEL
LIN {X 0,Y 492.428,Z 530.619,A -85,B 0,C 180,E1 -6551.27,E2 -6551.27} C_VEL
LIN {X 0,Y 491.776,Z 544.15,A -85,B 0,C 180,E1 -6552.106,E2 -6552.106} C_VEL
LIN {X 0,Y 491.052,Z 556.63,A -85,B 0,C 180,E1 -6553.046,E2 -6553.046} C_VEL
LIN {X 0,Y 490.47,Z 567.63,A -85,B 0,C 180,E1 -6554.033,E2 -6554.033} C_VEL
LIN {X 0,Y 489.807,Z 579.079,A -85,B 0,C 180,E1 -6555.245,E2 -6555.245} C_VEL
LIN {X 0,Y 489.294,Z 589.099,A -85,B 0,C 180,E1 -6556.503,E2 -6556.503} C_VEL
LIN {X 0,Y 488.796,Z 598.4,A -85,B 0,C 180,E1 -6557.882,E2 -6557.882} C_VEL
LIN {X 0,Y 488.5,Z 607.093,A -85,B 0,C 180,E1 -6559.431,E2 -6559.431} C_VEL
LIN {X 0,Y 488.222,Z 613.86,A -85,B 0,C 180,E1 -6560.889,E2 -6560.889} C_VEL
LIN {X 0,Y 488.062,Z 620.115,A -85,B 0,C 180,E1 -6562.554,E2 -6562.554} C_VEL
LIN {X 0,Y 487.968,Z 624.953,A -85,B 0,C 180,E1 -6564.214,E2 -6564.214} C_VEL
LIN {X 0,Y 487.892,Z 628.498,A -85,B 0,C 180,E1 -6565.87,E2 -6565.87} C_VEL
LIN {X 0,Y 487.904,Z 630.831,A -85,B 0,C 180,E1 -6567.524,E2 -6567.524} C_VEL
LIN {X 0,Y 487.831,Z 632.003,A -85,B 0,C 180,E1 -6569.175,E2 -6569.175} C_VEL
LIN {X 0,Y 487.831,Z 632.002,A -85,B 0,C 180,E1 -6570.826,E2 -6570.826} C_VEL
LIN {X 0,Y 487.904,Z 630.826,A -85,B 0,C 180,E1 -6572.477,E2 -6572.477} C_VEL
LIN {X 0,Y 487.892,Z 628.492,A -85,B 0,C 180,E1 -6574.131,E2 -6574.131} C_VEL
LIN {X 0,Y 487.964,Z 624.952,A -85,B 0,C 180,E1 -6575.787,E2 -6575.787} C_VEL
LIN {X 0,Y 488.063,Z 620.116,A -85,B 0,C 180,E1 -6577.447,E2 -6577.447} C_VEL
LIN {X 0,Y 488.223,Z 613.853,A -85,B 0,C 180,E1 -6579.111,E2 -6579.111} C_VEL
LIN {X 0,Y 488.58,Z 605.994,A -85,B 0,C 180,E1 -6580.778,E2 -6580.778} C_VEL
LIN {X 0,Y 488.836,Z 597.867,A -85,B 0,C 180,E1 -6582.206,E2 -6582.206} C_VEL
LIN {X 0,Y 489.396,Z 587.569,A -85,B 0,C 180,E1 -6583.707,E2 -6583.707} C_VEL
LIN {X 0,Y 489.877,Z 577.276,A -85,B 0,C 180,E1 -6584.966,E2 -6584.966} C_VEL
LIN {X 0,Y 490.626,Z 564.825,A -85,B 0,C 180,E1 -6586.24,E2 -6586.24} C_VEL
LIN {X 0,Y 491.346,Z 551.393,A -85,B 0,C 180,E1 -6587.373,E2 -6587.373} C_VEL
LIN {X 0,Y 492.124,Z 537.734,A -85,B 0,C 180,E1 -6588.312,E2 -6588.312} C_VEL
LIN {X 0,Y 492.753,Z 523.59,A -85,B 0,C 180,E1 -6589.096,E2 -6589.096} C_VEL
LIN {X 0,Y 493.41,Z 508.401,A -85,B 0,C 180,E1 -6589.743,E2 -6589.743} C_VEL
LIN {X 0,Y 493.896,Z 493.865,A -85,B 0,C 180,E1 -6590.194,E2 -6590.194} C_VEL
LIN {X 0,Y 494.205,Z 478.91,A -85,B 0,C 180,E1 -6590.499,E2 -6590.499} C_VEL
LIN {X 0,Y 495.495,Z 340.815,A -85,B 0,C 180,E1 -6592.549,E2 -6592.549} C_VEL
LIN {X 0,Y 491.524,Z 318.938,A -85,B 0,C 180,E1 -6593.104,E2 -6593.104} C_VEL
LIN {X 0,Y 492.38,Z 300.335,A -85,B 0,C 180,E1 -6595.66,E2 -6595.66} C_VEL
LIN {X 0,Y 492.801,Z 289.589,A -85,B 0,C 180,E1 -6597.153,E2 -6597.153} C_VEL
LIN {X 0,Y 489.387,Z 274.891,A -85,B 0,C 180,E1 -6599.463,E2 -6599.463} C_VEL
LIN {X 0,Y 488.742,Z 272.231,A -85,B 0,C 180,E1 -6599.921,E2 -6599.921} C_VEL
LIN {X 0,Y 488.737,Z 272.23,A -85,B 0,C 180,E1 -6603.485,E2 -6603.485} C_VEL
LIN {X 0,Y 488.685,Z 272.239,A -85,B 0,C 180,E1 -6606.355,E2 -6606.355} C_VEL
LIN {X 0,Y 488.703,Z 272.227,A -85,B 0,C 180,E1 -6609.255,E2 -6609.255} C_VEL
LIN {X 0,Y 488.69,Z 272.24,A -85,B 0,C 180,E1 -6612.526,E2 -6612.526} C_VEL
LIN {X 0,Y 488.704,Z 272.231,A -85,B 0,C 180,E1 -6615.198,E2 -6615.198} C_VEL
LIN {X 0,Y 488.711,Z 272.235,A -85,B 0,C 180,E1 -6618.585,E2 -6618.585} C_VEL
LIN {X 0,Y 488.704,Z 272.232,A -85,B 0,C 180,E1 -6620.948,E2 -6620.948} C_VEL
LIN {X 0,Y 488.673,Z 272.237,A -85,B 0,C 180,E1 -6623.868,E2 -6623.868} C_VEL
LIN {X 0,Y 488.742,Z 272.225,A -85,B 0,C 180,E1 -6626.878,E2 -6626.878} C_VEL
LIN {X 0,Y 488.728,Z 272.229,A -85,B 0,C 180,E1 -6629.781,E2 -6629.781} C_VEL
LIN {X 0,Y 488.718,Z 272.227,A -85,B 0,C 180,E1 -6633.075,E2 -6633.075} C_VEL
LIN {X 0,Y 488.679,Z 272.237,A -85,B 0,C 180,E1 -6636.254,E2 -6636.254} C_VEL
LIN {X 0,Y 488.751,Z 272.225,A -85,B 0,C 180,E1 -6639.176,E2 -6639.176} C_VEL
LIN {X 0,Y 488.752,Z 272.224,A -85,B 0,C 180,E1 -6641.632,E2 -6641.632} C_VEL
LIN {X 0,Y 488.766,Z 272.22,A -85,B 0,C 180,E1 -6645,E2 -6645} C_VEL
LIN {X 0,Y 488.81,Z 272.217,A -85,B 0,C 180,E1 -6648.388,E2 -6648.388} C_VEL
LIN {X 0,Y 488.767,Z 272.229,A -85,B 0,C 180,E1 -6651.733,E2 -6651.733} C_VEL
LIN {X 0,Y 488.82,Z 272.221,A -85,B 0,C 180,E1 -6654.224,E2 -6654.224} C_VEL
LIN {X 0,Y 488.947,Z 272.202,A -85,B 0,C 180,E1 -6657.529,E2 -6657.529} C_VEL
LIN {X 0,Y 488.945,Z 272.206,A -85,B 0,C 180,E1 -6660,E2 -6660} C_VEL
LIN {X 0,Y 488.954,Z 272.199,A -85,B 0,C 180,E1 -6662.471,E2 -6662.471} C_VEL
LIN {X 0,Y 488.81,Z 272.221,A -85,B 0,C 180,E1 -6665.776,E2 -6665.776} C_VEL
LIN {X 0,Y 488.763,Z 272.225,A -85,B 0,C 180,E1 -6668.267,E2 -6668.267} C_VEL
LIN {X 0,Y 488.809,Z 272.222,A -85,B 0,C 180,E1 -6671.612,E2 -6671.612} C_VEL
LIN {X 0,Y 488.75,Z 272.222,A -85,B 0,C 180,E1 -6675.001,E2 -6675.001} C_VEL
LIN {X 0,Y 488.71,Z 272.227,A -85,B 0,C 180,E1 -6678.444,E2 -6678.444} C_VEL
LIN {X 0,Y 488.694,Z 272.234,A -85,B 0,C 180,E1 -6681.071,E2 -6681.071} C_VEL
LIN {X 0,Y 488.664,Z 272.242,A -85,B 0,C 180,E1 -6683.747,E2 -6683.747} C_VEL
LIN {X 0,Y 488.672,Z 272.231,A -85,B 0,C 180,E1 -6686.477,E2 -6686.477} C_VEL
LIN {X 0,Y 488.663,Z 272.232,A -85,B 0,C 180,E1 -6689.274,E2 -6689.274} C_VEL
LIN {X 0,Y 488.682,Z 272.233,A -85,B 0,C 180,E1 -6692.149,E2 -6692.149} C_VEL
LIN {X 0,Y 488.698,Z 272.236,A -85,B 0,C 180,E1 -6695.117,E2 -6695.117} C_VEL
LIN {X 0,Y 488.647,Z 272.237,A -85,B 0,C 180,E1 -6698.203,E2 -6698.203} C_VEL
LIN {X 0,Y 488.645,Z 272.243,A -85,B 0,C 180,E1 -6701.422,E2 -6701.422} C_VEL
LIN {X 0,Y 488.682,Z 272.235,A -85,B 0,C 180,E1 -6704.805,E2 -6704.805} C_VEL
LIN {X 0,Y 488.646,Z 272.242,A -85,B 0,C 180,E1 -6707.469,E2 -6707.469} C_VEL
LIN {X 0,Y 488.667,Z 272.237,A -85,B 0,C 180,E1 -6710.742,E2 -6710.742} C_VEL
LIN {X 0,Y 488.639,Z 272.241,A -85,B 0,C 180,E1 -6713.864,E2 -6713.864} C_VEL
LIN {X 0,Y 488.694,Z 272.232,A -85,B 0,C 180,E1 -6716.523,E2 -6716.523} C_VEL
LIN {X 0,Y 488.653,Z 272.241,A -85,B 0,C 180,E1 -6719.649,E2 -6719.649} C_VEL
LIN {X 0,Y 488.676,Z 272.238,A -85,B 0,C 180,E1 -6722.599,E2 -6722.599} C_VEL
LIN {X 0,Y 488.683,Z 272.238,A -85,B 0,C 180,E1 -6724.299,E2 -6724.299} C_VEL
LIN {X 0,Y 488.459,Z 273.02,A -85,B 0,C 180,E1 -6724.605,E2 -6724.605} C_VEL
LIN {X 0,Y 487.06,Z 276.3,A -85,B 0,C 180,E1 -6725.117,E2 -6725.117} C_VEL
LIN {X 0,Y 484.322,Z 281.986,A -85,B 0,C 180,E1 -6725.925,E2 -6725.925} C_VEL
LIN {X 0,Y 484.154,Z 284.19,A -85,B 0,C 180,E1 -6726.305,E2 -6726.305} C_VEL
LIN {X 0,Y 484.547,Z 286.197,A -85,B 0,C 180,E1 -6726.638,E2 -6726.638} C_VEL
LIN {X 0,Y 486.63,Z 293.236,A -85,B 0,C 180,E1 -6726.856,E2 -6726.856} C_VEL
LIN {X 0,Y 489.148,Z 303.755,A -85,B 0,C 180,E1 -6727.149,E2 -6727.149} C_VEL
LIN {X 0,Y 487.99,Z 416.074,A -85,B 0,C 180,E1 -6728.841,E2 -6728.841} C_VEL
LIN {X 0,Y 487.641,Z 451.08,A -85,B 0,C 180,E1 -6729.391,E2 -6729.391} C_VEL
LIN {X 0,Y 487.265,Z 466.464,A -85,B 0,C 180,E1 -6729.796,E2 -6729.796} C_VEL
LIN {X 0,Y 486.749,Z 480.945,A -85,B 0,C 180,E1 -6730.343,E2 -6730.343} C_VEL
LIN {X 0,Y 486.117,Z 494.5,A -85,B 0,C 180,E1 -6731.016,E2 -6731.016} C_VEL
LIN {X 0,Y 485.469,Z 508.079,A -85,B 0,C 180,E1 -6731.865,E2 -6731.865} C_VEL
LIN {X 0,Y 484.719,Z 520.561,A -85,B 0,C 180,E1 -6732.817,E2 -6732.817} C_VEL
LIN {X 0,Y 483.956,Z 533.192,A -85,B 0,C 180,E1 -6733.983,E2 -6733.983} C_VEL
LIN {X 0,Y 483.251,Z 544.637,A -85,B 0,C 180,E1 -6735.255,E2 -6735.255} C_VEL
LIN {X 0,Y 482.612,Z 554.266,A -85,B 0,C 180,E1 -6736.526,E2 -6736.526} C_VEL
LIN {X 0,Y 482.099,Z 563.579,A -85,B 0,C 180,E1 -6737.989,E2 -6737.989} C_VEL
LIN {X 0,Y 481.65,Z 571.545,A -85,B 0,C 180,E1 -6739.49,E2 -6739.49} C_VEL
LIN {X 0,Y 481.339,Z 578.868,A -85,B 0,C 180,E1 -6741.181,E2 -6741.181} C_VEL
LIN {X 0,Y 481.081,Z 584.68,A -85,B 0,C 180,E1 -6742.866,E2 -6742.866} C_VEL
LIN {X 0,Y 481.069,Z 588.116,A -85,B 0,C 180,E1 -6744.13,E2 -6744.13} C_VEL
LIN {X 0,Y 480.9,Z 591.606,A -85,B 0,C 180,E1 -6745.809,E2 -6745.809} C_VEL
LIN {X 0,Y 480.865,Z 593.914,A -85,B 0,C 180,E1 -6747.487,E2 -6747.487} C_VEL
LIN {X 0,Y 480.757,Z 595.099,A -85,B 0,C 180,E1 -6749.162,E2 -6749.162} C_VEL
LIN {X 0,Y 480.758,Z 595.117,A -85,B 0,C 180,E1 -6750.837,E2 -6750.837} C_VEL
LIN {X 0,Y 480.866,Z 594.004,A -85,B 0,C 180,E1 -6752.513,E2 -6752.513} C_VEL
LIN {X 0,Y 480.899,Z 591.766,A -85,B 0,C 180,E1 -6754.19,E2 -6754.19} C_VEL
LIN {X 0,Y 481.06,Z 588.342,A -85,B 0,C 180,E1 -6755.869,E2 -6755.869} C_VEL
LIN {X 0,Y 481.143,Z 583.659,A -85,B 0,C 180,E1 -6757.554,E2 -6757.554} C_VEL
LIN {X 0,Y 481.384,Z 577.586,A -85,B 0,C 180,E1 -6759.241,E2 -6759.241} C_VEL
LIN {X 0,Y 481.773,Z 569.934,A -85,B 0,C 180,E1 -6760.931,E2 -6760.931} C_VEL
LIN {X 0,Y 482.158,Z 561.754,A -85,B 0,C 180,E1 -6762.418,E2 -6762.418} C_VEL
LIN {X 0,Y 482.822,Z 551.937,A -85,B 0,C 180,E1 -6763.897,E2 -6763.897} C_VEL
LIN {X 0,Y 483.434,Z 541.848,A -85,B 0,C 180,E1 -6765.169,E2 -6765.169} C_VEL
LIN {X 0,Y 484.141,Z 530.178,A -85,B 0,C 180,E1 -6766.408,E2 -6766.408} C_VEL
LIN {X 0,Y 484.879,Z 517.782,A -85,B 0,C 180,E1 -6767.503,E2 -6767.503} C_VEL
LIN {X 0,Y 485.681,Z 504.681,A -85,B 0,C 180,E1 -6768.453,E2 -6768.453} C_VEL
LIN {X 0,Y 486.24,Z 492.203,A -85,B 0,C 180,E1 -6769.197,E2 -6769.197} C_VEL
LIN {X 0,Y 486.893,Z 477.664,A -85,B 0,C 180,E1 -6769.88,E2 -6769.88} C_VEL
LIN {X 0,Y 487.314,Z 462.993,A -85,B 0,C 180,E1 -6770.399,E2 -6770.399} C_VEL
LIN {X 0,Y 487.662,Z 448.22,A -85,B 0,C 180,E1 -6770.753,E2 -6770.753} C_VEL
LIN {X 0,Y 489.076,Z 314.944,A -85,B 0,C 180,E1 -6772.771,E2 -6772.771} C_VEL
LIN {X 0,Y 489.005,Z 303.295,A -85,B 0,C 180,E1 -6772.957,E2 -6772.957} C_VEL
LIN {X 0,Y 485.362,Z 288.4,A -85,B 0,C 180,E1 -6773.377,E2 -6773.377} C_VEL
LIN {X 0,Y 484.495,Z 285.911,A -85,B 0,C 180,E1 -6773.474,E2 -6773.474} C_VEL
LIN {X 0,Y 481.646,Z 273.114,A -85,B 0,C 180,E1 -6775.915,E2 -6775.915} C_VEL
LIN {X 0,Y 481.63,Z 273.12,A -85,B 0,C 180,E1 -6778.892,E2 -6778.892} C_VEL
LIN {X 0,Y 481.63,Z 273.118,A -85,B 0,C 180,E1 -6782.184,E2 -6782.184} C_VEL
LIN {X 0,Y 481.647,Z 273.114,A -85,B 0,C 180,E1 -6785.201,E2 -6785.201} C_VEL
LIN {X 0,Y 481.629,Z 273.115,A -85,B 0,C 180,E1 -6788.003,E2 -6788.003} C_VEL
LIN {X 0,Y 481.621,Z 273.119,A -85,B 0,C 180,E1 -6791.045,E2 -6791.045} C_VEL
LIN {X 0,Y 481.648,Z 273.11,A -85,B 0,C 180,E1 -6794.458,E2 -6794.458} C_VEL
LIN {X 0,Y 481.609,Z 273.113,A -85,B 0,C 180,E1 -6796.856,E2 -6796.856} C_VEL
LIN {X 0,Y 481.625,Z 273.113,A -85,B 0,C 180,E1 -6800.054,E2 -6800.054} C_VEL
LIN {X 0,Y 481.598,Z 273.105,A -85,B 0,C 180,E1 -6803.25,E2 -6803.25} C_VEL
LIN {X 0,Y 481.669,Z 273.109,A -85,B 0,C 180,E1 -6806.327,E2 -6806.327} C_VEL
LIN {X 0,Y 481.608,Z 273.114,A -85,B 0,C 180,E1 -6809.426,E2 -6809.426} C_VEL
LIN {X 0,Y 481.641,Z 273.113,A -85,B 0,C 180,E1 -6812.164,E2 -6812.164} C_VEL
LIN {X 0,Y 481.667,Z 273.11,A -85,B 0,C 180,E1 -6814.967,E2 -6814.967} C_VEL
LIN {X 0,Y 481.631,Z 273.11,A -85,B 0,C 180,E1 -6817.704,E2 -6817.704} C_VEL
LIN {X 0,Y 481.655,Z 273.113,A -85,B 0,C 180,E1 -6820.391,E2 -6820.391} C_VEL
LIN {X 0,Y 481.612,Z 273.116,A -85,B 0,C 180,E1 -6823.031,E2 -6823.031} C_VEL
LIN {X 0,Y 481.665,Z 273.105,A -85,B 0,C 180,E1 -6825.638,E2 -6825.638} C_VEL
LIN {X 0,Y 481.749,Z 273.103,A -85,B 0,C 180,E1 -6828.215,E2 -6828.215} C_VEL
LIN {X 0,Y 481.716,Z 273.098,A -85,B 0,C 180,E1 -6831.611,E2 -6831.611} C_VEL
LIN {X 0,Y 481.765,Z 273.102,A -85,B 0,C 180,E1 -6834.139,E2 -6834.139} C_VEL
LIN {X 0,Y 481.915,Z 273.076,A -85,B 0,C 180,E1 -6837.492,E2 -6837.492} C_VEL
LIN {X 0,Y 481.845,Z 273.081,A -85,B 0,C 180,E1 -6840.836,E2 -6840.836} C_VEL
LIN {X 0,Y 481.913,Z 273.081,A -85,B 0,C 180,E1 -6842.507,E2 -6842.507} C_VEL
LIN {X 0,Y 481.785,Z 273.095,A -85,B 0,C 180,E1 -6845.861,E2 -6845.861} C_VEL
LIN {X 0,Y 481.727,Z 273.104,A -85,B 0,C 180,E1 -6848.389,E2 -6848.389} C_VEL
LIN {X 0,Y 481.749,Z 273.098,A -85,B 0,C 180,E1 -6851.785,E2 -6851.785} C_VEL
LIN {X 0,Y 481.741,Z 273.095,A -85,B 0,C 180,E1 -6855.224,E2 -6855.224} C_VEL
LIN {X 0,Y 481.706,Z 273.101,A -85,B 0,C 180,E1 -6858.722,E2 -6858.722} C_VEL
LIN {X 0,Y 481.644,Z 273.113,A -85,B 0,C 180,E1 -6861.395,E2 -6861.395} C_VEL
LIN {X 0,Y 481.655,Z 273.102,A -85,B 0,C 180,E1 -6864.114,E2 -6864.114} C_VEL
LIN {X 0,Y 481.693,Z 273.101,A -85,B 0,C 180,E1 -6867.127,E2 -6867.127} C_VEL
LIN {X 0,Y 481.671,Z 273.112,A -85,B 0,C 180,E1 -6869.741,E2 -6869.741} C_VEL
LIN {X 0,Y 481.67,Z 273.101,A -85,B 0,C 180,E1 -6872.674,E2 -6872.674} C_VEL
LIN {X 0,Y 481.636,Z 273.116,A -85,B 0,C 180,E1 -6875.709,E2 -6875.709} C_VEL
LIN {X 0,Y 481.669,Z 273.105,A -85,B 0,C 180,E1 -6878.859,E2 -6878.859} C_VEL
LIN {X 0,Y 481.651,Z 273.115,A -85,B 0,C 180,E1 -6881.913,E2 -6881.913} C_VEL
LIN {X 0,Y 481.653,Z 273.109,A -85,B 0,C 180,E1 -6884.458,E2 -6884.458} C_VEL
LIN {X 0,Y 481.646,Z 273.113,A -85,B 0,C 180,E1 -6887.839,E2 -6887.839} C_VEL
LIN {X 0,Y 481.678,Z 273.107,A -85,B 0,C 180,E1 -6890.651,E2 -6890.651} C_VEL
LIN {X 0,Y 481.629,Z 273.119,A -85,B 0,C 180,E1 -6893.376,E2 -6893.376} C_VEL
LIN {X 0,Y 481.709,Z 273.104,A -85,B 0,C 180,E1 -6896.33,E2 -6896.33} C_VEL
LIN {X 0,Y 481.706,Z 273.217,A -85,B 0,C 180,E1 -6899.809,E2 -6899.809} C_VEL
LIN {X 0,Y 485.426,Z 288.523,A -85,B 0,C 180,E1 -6902.283,E2 -6902.283} C_VEL
LIN {X 0,Y 486.027,Z 292.59,A -85,B 0,C 180,E1 -6902.904,E2 -6902.904} C_VEL
LIN {X 0,Y 485.039,Z 313.045,A -85,B 0,C 180,E1 -6905.77,E2 -6905.77} C_VEL
LIN {X 0,Y 484.668,Z 318.847,A -85,B 0,C 180,E1 -6906.575,E2 -6906.575} C_VEL
LIN {X 0,Y 488.95,Z 341.254,A -85,B 0,C 180,E1 -6907.142,E2 -6907.142} C_VEL
LIN {X 0,Y 487.463,Z 484.722,A -85,B 0,C 180,E1 -6909.315,E2 -6909.315} C_VEL
LIN {X 0,Y 487.011,Z 500.316,A -85,B 0,C 180,E1 -6909.709,E2 -6909.709} C_VEL
LIN {X 0,Y 486.389,Z 515.762,A -85,B 0,C 180,E1 -6910.279,E2 -6910.279} C_VEL
LIN {X 0,Y 485.667,Z 530.349,A -85,B 0,C 180,E1 -6910.999,E2 -6910.999} C_VEL
LIN {X 0,Y 484.966,Z 543.879,A -85,B 0,C 180,E1 -6911.846,E2 -6911.846} C_VEL
LIN {X 0,Y 484.22,Z 556.359,A -85,B 0,C 180,E1 -6912.799,E2 -6912.799} C_VEL
LIN {X 0,Y 483.521,Z 567.813,A -85,B 0,C 180,E1 -6913.843,E2 -6913.843} C_VEL
LIN {X 0,Y 482.845,Z 578.805,A -85,B 0,C 180,E1 -6915.028,E2 -6915.028} C_VEL
LIN {X 0,Y 482.329,Z 588.826,A -85,B 0,C 180,E1 -6916.304,E2 -6916.304} C_VEL
LIN {X 0,Y 481.744,Z 598.735,A -85,B 0,C 180,E1 -6917.806,E2 -6917.806} C_VEL
LIN {X 0,Y 481.471,Z 606.82,A -85,B 0,C 180,E1 -6919.274,E2 -6919.274} C_VEL
LIN {X 0,Y 481.149,Z 613.587,A -85,B 0,C 180,E1 -6920.754,E2 -6920.754} C_VEL
LIN {X 0,Y 480.986,Z 619.843,A -85,B 0,C 180,E1 -6922.444,E2 -6922.444} C_VEL
LIN {X 0,Y 480.876,Z 624.682,A -85,B 0,C 180,E1 -6924.128,E2 -6924.128} C_VEL
LIN {X 0,Y 480.795,Z 628.226,A -85,B 0,C 180,E1 -6925.809,E2 -6925.809} C_VEL
LIN {X 0,Y 480.818,Z 630.561,A -85,B 0,C 180,E1 -6927.487,E2 -6927.487} C_VEL
LIN {X 0,Y 480.757,Z 631.733,A -85,B 0,C 180,E1 -6929.163,E2 -6929.163} C_VEL
LIN {X 0,Y 480.757,Z 631.732,A -85,B 0,C 180,E1 -6930.838,E2 -6930.838} C_VEL
LIN {X 0,Y 480.818,Z 630.556,A -85,B 0,C 180,E1 -6932.514,E2 -6932.514} C_VEL
LIN {X 0,Y 480.795,Z 628.221,A -85,B 0,C 180,E1 -6934.192,E2 -6934.192} C_VEL
LIN {X 0,Y 480.87,Z 624.681,A -85,B 0,C 180,E1 -6935.872,E2 -6935.872} C_VEL
LIN {X 0,Y 480.987,Z 619.844,A -85,B 0,C 180,E1 -6937.557,E2 -6937.557} C_VEL
LIN {X 0,Y 481.15,Z 613.58,A -85,B 0,C 180,E1 -6939.246,E2 -6939.246} C_VEL
LIN {X 0,Y 481.551,Z 605.721,A -85,B 0,C 180,E1 -6940.937,E2 -6940.937} C_VEL
LIN {X 0,Y 481.796,Z 597.913,A -85,B 0,C 180,E1 -6942.334,E2 -6942.334} C_VEL
LIN {X 0,Y 482.386,Z 587.294,A -85,B 0,C 180,E1 -6943.91,E2 -6943.91} C_VEL
LIN {X 0,Y 482.943,Z 577.002,A -85,B 0,C 180,E1 -6945.186,E2 -6945.186} C_VEL
LIN {X 0,Y 483.769,Z 564.308,A -85,B 0,C 180,E1 -6946.5,E2 -6946.5} C_VEL
LIN {X 0,Y 484.521,Z 551.118,A -85,B 0,C 180,E1 -6947.626,E2 -6947.626} C_VEL
LIN {X 0,Y 485.322,Z 537.458,A -85,B 0,C 180,E1 -6948.578,E2 -6948.578} C_VEL
LIN {X 0,Y 486.018,Z 523.314,A -85,B 0,C 180,E1 -6949.372,E2 -6949.372} C_VEL
LIN {X 0,Y 486.688,Z 507.89,A -85,B 0,C 180,E1 -6950.036,E2 -6950.036} C_VEL
LIN {X 0,Y 487.246,Z 492.855,A -85,B 0,C 180,E1 -6950.502,E2 -6950.502} C_VEL
LIN {X 0,Y 487.558,Z 476.938,A -85,B 0,C 180,E1 -6950.819,E2 -6950.819} C_VEL
LIN {X 0,Y 488.925,Z 341.507,A -85,B 0,C 180,E1 -6952.854,E2 -6952.854} C_VEL
LIN {X 0,Y 484.705,Z 318.833,A -85,B 0,C 180,E1 -6953.424,E2 -6953.424} C_VEL
LIN {X 0,Y 485.583,Z 301.037,A -85,B 0,C 180,E1 -6955.907,E2 -6955.907} C_VEL
LIN {X 0,Y 485.956,Z 290.943,A -85,B 0,C 180,E1 -6957.334,E2 -6957.334} C_VEL
LIN {X 0,Y 482.054,Z 274.613,A -85,B 0,C 180,E1 -6959.957,E2 -6959.957} C_VEL
LIN {X 0,Y 481.694,Z 273.109,A -85,B 0,C 180,E1 -6960.223,E2 -6960.223} C_VEL
LIN {X 0,Y 481.699,Z 273.107,A -85,B 0,C 180,E1 -6963.734,E2 -6963.734} C_VEL
LIN {X 0,Y 481.628,Z 273.118,A -85,B 0,C 180,E1 -6966.747,E2 -6966.747} C_VEL
LIN {X 0,Y 481.67,Z 273.104,A -85,B 0,C 180,E1 -6969.942,E2 -6969.942} C_VEL
LIN {X 0,Y 481.629,Z 273.113,A -85,B 0,C 180,E1 -6973.147,E2 -6973.147} C_VEL
LIN {X 0,Y 481.657,Z 273.109,A -85,B 0,C 180,E1 -6975.642,E2 -6975.642} C_VEL
LIN {X 0,Y 481.66,Z 273.109,A -85,B 0,C 180,E1 -6978.959,E2 -6978.959} C_VEL
LIN {X 0,Y 481.653,Z 273.113,A -85,B 0,C 180,E1 -6981.994,E2 -6981.994} C_VEL
LIN {X 0,Y 481.691,Z 273.102,A -85,B 0,C 180,E1 -6985.318,E2 -6985.318} C_VEL
LIN {X 0,Y 481.65,Z 273.114,A -85,B 0,C 180,E1 -6988.312,E2 -6988.312} C_VEL
LIN {X 0,Y 481.678,Z 273.103,A -85,B 0,C 180,E1 -6991.217,E2 -6991.217} C_VEL
LIN {X 0,Y 481.66,Z 273.111,A -85,B 0,C 180,E1 -6994.041,E2 -6994.041} C_VEL
LIN {X 0,Y 481.679,Z 273.103,A -85,B 0,C 180,E1 -6996.812,E2 -6996.812} C_VEL
LIN {X 0,Y 481.7,Z 273.105,A -85,B 0,C 180,E1 -6999.503,E2 -6999.503} C_VEL
LIN {X 0,Y 481.693,Z 273.112,A -85,B 0,C 180,E1 -7002.158,E2 -7002.158} C_VEL
LIN {X 0,Y 481.747,Z 273.095,A -85,B 0,C 180,E1 -7004.776,E2 -7004.776} C_VEL
LIN {X 0,Y 481.756,Z 273.098,A -85,B 0,C 180,E1 -7008.215,E2 -7008.215} C_VEL
LIN {X 0,Y 481.726,Z 273.104,A -85,B 0,C 180,E1 -7011.611,E2 -7011.611} C_VEL
LIN {X 0,Y 481.781,Z 273.099,A -85,B 0,C 180,E1 -7014.139,E2 -7014.139} C_VEL
LIN {X 0,Y 481.912,Z 273.077,A -85,B 0,C 180,E1 -7017.493,E2 -7017.493} C_VEL
LIN {X 0,Y 481.914,Z 273.081,A -85,B 0,C 180,E1 -7020,E2 -7020} C_VEL
LIN {X 0,Y 481.921,Z 273.075,A -85,B 0,C 180,E1 -7022.508,E2 -7022.508} C_VEL
LIN {X 0,Y 481.771,Z 273.097,A -85,B 0,C 180,E1 -7025.861,E2 -7025.861} C_VEL
LIN {X 0,Y 481.722,Z 273.102,A -85,B 0,C 180,E1 -7028.389,E2 -7028.389} C_VEL
LIN {X 0,Y 481.755,Z 273.103,A -85,B 0,C 180,E1 -7031.785,E2 -7031.785} C_VEL
LIN {X 0,Y 481.733,Z 273.098,A -85,B 0,C 180,E1 -7035.225,E2 -7035.225} C_VEL
LIN {X 0,Y 481.654,Z 273.106,A -85,B 0,C 180,E1 -7038.724,E2 -7038.724} C_VEL
LIN {X 0,Y 481.634,Z 273.118,A -85,B 0,C 180,E1 -7041.395,E2 -7041.395} C_VEL
LIN {X 0,Y 481.644,Z 273.112,A -85,B 0,C 180,E1 -7044.115,E2 -7044.115} C_VEL
LIN {X 0,Y 481.646,Z 273.11,A -85,B 0,C 180,E1 -7047.114,E2 -7047.114} C_VEL
LIN {X 0,Y 481.604,Z 273.119,A -85,B 0,C 180,E1 -7049.746,E2 -7049.746} C_VEL
LIN {X 0,Y 481.637,Z 273.111,A -85,B 0,C 180,E1 -7052.677,E2 -7052.677} C_VEL
LIN {X 0,Y 481.642,Z 273.116,A -85,B 0,C 180,E1 -7055.2,E2 -7055.2} C_VEL
LIN {X 0,Y 481.623,Z 273.113,A -85,B 0,C 180,E1 -7058.001,E2 -7058.001} C_VEL
LIN {X 0,Y 481.606,Z 273.119,A -85,B 0,C 180,E1 -7061.047,E2 -7061.047} C_VEL
LIN {X 0,Y 481.623,Z 273.112,A -85,B 0,C 180,E1 -7064.462,E2 -7064.462} C_VEL
LIN {X 0,Y 481.608,Z 273.115,A -85,B 0,C 180,E1 -7067.834,E2 -7067.834} C_VEL
LIN {X 0,Y 481.631,Z 273.113,A -85,B 0,C 180,E1 -7070.659,E2 -7070.659} C_VEL
LIN {X 0,Y 481.603,Z 273.119,A -85,B 0,C 180,E1 -7073.38,E2 -7073.38} C_VEL
LIN {X 0,Y 481.673,Z 273.106,A -85,B 0,C 180,E1 -7076.327,E2 -7076.327} C_VEL
LIN {X 0,Y 481.612,Z 273.121,A -85,B 0,C 180,E1 -7079.425,E2 -7079.425} C_VEL
LIN {X 0,Y 481.643,Z 273.113,A -85,B 0,C 180,E1 -7082.164,E2 -7082.164} C_VEL
LIN {X 0,Y 481.642,Z 273.172,A -85,B 0,C 180,E1 -7084.229,E2 -7084.229} C_VEL
LIN {X 0,Y 484.154,Z 284.19,A -85,B 0,C 180,E1 -7086.305,E2 -7086.305} C_VEL
LIN {X 0,Y 484.72,Z 286.191,A -85,B 0,C 180,E1 -7086.545,E2 -7086.545} C_VEL
LIN {X 0,Y 485.346,Z 289.225,A -85,B 0,C 180,E1 -7086.713,E2 -7086.713} C_VEL
LIN {X 0,Y 485.22,Z 291.688,A -85,B 0,C 180,E1 -7086.759,E2 -7086.759} C_VEL
LIN {X 0,Y 482.757,Z 300.351,A -85,B 0,C 180,E1 -7086.769,E2 -7086.769} C_VEL
LIN {X 0,Y 482.477,Z 304.214,A -85,B 0,C 180,E1 -7086.817,E2 -7086.817} C_VEL
LIN {X 0,Y 482.616,Z 304.958,A -85,B 0,C 180,E1 -7086.836,E2 -7086.836} C_VEL
LIN {X 0,Y 481.399,Z 416.374,A -85,B 0,C 180,E1 -7088.537,E2 -7088.537} C_VEL
LIN {X 0,Y 481.017,Z 451.37,A -85,B 0,C 180,E1 -7089.094,E2 -7089.094} C_VEL
LIN {X 0,Y 480.62,Z 466.595,A -85,B 0,C 180,E1 -7089.499,E2 -7089.499} C_VEL
LIN {X 0,Y 480.078,Z 481.381,A -85,B 0,C 180,E1 -7090.066,E2 -7090.066} C_VEL
LIN {X 0,Y 479.411,Z 494.779,A -85,B 0,C 180,E1 -7090.74,E2 -7090.74} C_VEL
LIN {X 0,Y 478.733,Z 508.356,A -85,B 0,C 180,E1 -7091.601,E2 -7091.601} C_VEL
LIN {X 0,Y 477.919,Z 520.838,A -85,B 0,C 180,E1 -7092.565,E2 -7092.565} C_VEL
LIN {X 0,Y 477.117,Z 533.468,A -85,B 0,C 180,E1 -7093.747,E2 -7093.747} C_VEL
LIN {X 0,Y 476.352,Z 544.913,A -85,B 0,C 180,E1 -7095.037,E2 -7095.037} C_VEL
LIN {X 0,Y 475.695,Z 554.541,A -85,B 0,C 180,E1 -7096.326,E2 -7096.326} C_VEL
LIN {X 0,Y 475.109,Z 564.067,A -85,B 0,C 180,E1 -7097.848,E2 -7097.848} C_VEL
LIN {X 0,Y 474.654,Z 571.819,A -85,B 0,C 180,E1 -7099.334,E2 -7099.334} C_VEL
LIN {X 0,Y 474.297,Z 579.142,A -85,B 0,C 180,E1 -7101.049,E2 -7101.049} C_VEL
LIN {X 0,Y 474.014,Z 584.953,A -85,B 0,C 180,E1 -7102.76,E2 -7102.76} C_VEL
LIN {X 0,Y 473.983,Z 588.388,A -85,B 0,C 180,E1 -7104.042,E2 -7104.042} C_VEL
LIN {X 0,Y 473.806,Z 591.878,A -85,B 0,C 180,E1 -7105.746,E2 -7105.746} C_VEL
LIN {X 0,Y 473.78,Z 594.185,A -85,B 0,C 180,E1 -7107.449,E2 -7107.449} C_VEL
LIN {X 0,Y 473.686,Z 595.369,A -85,B 0,C 180,E1 -7109.149,E2 -7109.149} C_VEL
LIN {X 0,Y 473.686,Z 595.386,A -85,B 0,C 180,E1 -7110.85,E2 -7110.85} C_VEL
LIN {X 0,Y 473.78,Z 594.273,A -85,B 0,C 180,E1 -7112.55,E2 -7112.55} C_VEL
LIN {X 0,Y 473.805,Z 592.036,A -85,B 0,C 180,E1 -7114.253,E2 -7114.253} C_VEL
LIN {X 0,Y 473.975,Z 588.612,A -85,B 0,C 180,E1 -7115.957,E2 -7115.957} C_VEL
LIN {X 0,Y 474.09,Z 583.928,A -85,B 0,C 180,E1 -7117.667,E2 -7117.667} C_VEL
LIN {X 0,Y 474.337,Z 577.855,A -85,B 0,C 180,E1 -7119.38,E2 -7119.38} C_VEL
LIN {X 0,Y 474.794,Z 570.202,A -85,B 0,C 180,E1 -7121.094,E2 -7121.094} C_VEL
LIN {X 0,Y 475.169,Z 562.438,A -85,B 0,C 180,E1 -7122.532,E2 -7122.532} C_VEL
LIN {X 0,Y 475.901,Z 552.205,A -85,B 0,C 180,E1 -7124.103,E2 -7124.103} C_VEL
LIN {X 0,Y 476.563,Z 542.116,A -85,B 0,C 180,E1 -7125.393,E2 -7125.393} C_VEL
LIN {X 0,Y 477.307,Z 530.788,A -85,B 0,C 180,E1 -7126.614,E2 -7126.614} C_VEL
LIN {X 0,Y 478.098,Z 518.048,A -85,B 0,C 180,E1 -7127.759,E2 -7127.759} C_VEL
LIN {X 0,Y 478.954,Z 504.944,A -85,B 0,C 180,E1 -7128.722,E2 -7128.722} C_VEL
LIN {X 0,Y 479.56,Z 492.464,A -85,B 0,C 180,E1 -7129.475,E2 -7129.475} C_VEL
LIN {X 0,Y 480.251,Z 477.176,A -85,B 0,C 180,E1 -7130.199,E2 -7130.199} C_VEL
LIN {X 0,Y 480.727,Z 462.251,A -85,B 0,C 180,E1 -7130.721,E2 -7130.721} C_VEL
LIN {X 0,Y 481.088,Z 446.811,A -85,B 0,C 180,E1 -7131.081,E2 -7131.081} C_VEL
LIN {X 0,Y 482.509,Z 319.226,A -85,B 0,C 180,E1 -7133.035,E2 -7133.035} C_VEL
LIN {X 0,Y 482.494,Z 304.504,A -85,B 0,C 180,E1 -7133.27,E2 -7133.27} C_VEL
LIN {X 0,Y 479.033,Z 290.604,A -85,B 0,C 180,E1 -7133.673,E2 -7133.673} C_VEL
LIN {X 0,Y 477.338,Z 286.103,A -85,B 0,C 180,E1 -7133.862,E2 -7133.862} C_VEL
LIN {X 0,Y 474.618,Z 273.99,A -85,B 0,C 180,E1 -7136.201,E2 -7136.201} C_VEL
LIN {X 0,Y 474.592,Z 273.997,A -85,B 0,C 180,E1 -7139.254,E2 -7139.254} C_VEL
LIN {X 0,Y 474.582,Z 273.998,A -85,B 0,C 180,E1 -7142.424,E2 -7142.424} C_VEL
LIN {X 0,Y 474.598,Z 273.989,A -85,B 0,C 180,E1 -7145.466,E2 -7145.466} C_VEL
LIN {X 0,Y 474.587,Z 273.995,A -85,B 0,C 180,E1 -7148.459,E2 -7148.459} C_VEL
LIN {X 0,Y 474.597,Z 273.995,A -85,B 0,C 180,E1 -7150.955,E2 -7150.955} C_VEL
LIN {X 0,Y 474.577,Z 273.988,A -85,B 0,C 180,E1 -7154.108,E2 -7154.108} C_VEL
LIN {X 0,Y 474.563,Z 273.988,A -85,B 0,C 180,E1 -7157.06,E2 -7157.06} C_VEL
LIN {X 0,Y 474.595,Z 273.992,A -85,B 0,C 180,E1 -7160.449,E2 -7160.449} C_VEL
LIN {X 0,Y 474.563,Z 273.979,A -85,B 0,C 180,E1 -7163.674,E2 -7163.674} C_VEL
LIN {X 0,Y 474.605,Z 273.994,A -85,B 0,C 180,E1 -7166.777,E2 -7166.777} C_VEL
LIN {X 0,Y 474.547,Z 273.994,A -85,B 0,C 180,E1 -7169.766,E2 -7169.766} C_VEL
LIN {X 0,Y 474.6,Z 273.991,A -85,B 0,C 180,E1 -7172.684,E2 -7172.684} C_VEL
LIN {X 0,Y 474.619,Z 273.985,A -85,B 0,C 180,E1 -7175.505,E2 -7175.505} C_VEL
LIN {X 0,Y 474.637,Z 273.984,A -85,B 0,C 180,E1 -7179.184,E2 -7179.184} C_VEL
LIN {X 0,Y 474.616,Z 273.983,A -85,B 0,C 180,E1 -7181.883,E2 -7181.883} C_VEL
LIN {X 0,Y 474.686,Z 273.98,A -85,B 0,C 180,E1 -7184.544,E2 -7184.544} C_VEL
LIN {X 0,Y 474.703,Z 273.978,A -85,B 0,C 180,E1 -7188.037,E2 -7188.037} C_VEL
LIN {X 0,Y 474.665,Z 273.975,A -85,B 0,C 180,E1 -7191.485,E2 -7191.485} C_VEL
LIN {X 0,Y 474.728,Z 273.977,A -85,B 0,C 180,E1 -7194.052,E2 -7194.052} C_VEL
LIN {X 0,Y 474.881,Z 273.952,A -85,B 0,C 180,E1 -7197.455,E2 -7197.455} C_VEL
LIN {X 0,Y 474.878,Z 273.958,A -85,B 0,C 180,E1 -7200,E2 -7200} C_VEL
LIN {X 0,Y 474.878,Z 273.956,A -85,B 0,C 180,E1 -7202.545,E2 -7202.545} C_VEL
LIN {X 0,Y 474.747,Z 273.971,A -85,B 0,C 180,E1 -7205.948,E2 -7205.948} C_VEL
LIN {X 0,Y 474.702,Z 273.978,A -85,B 0,C 180,E1 -7208.514,E2 -7208.514} C_VEL
LIN {X 0,Y 474.703,Z 273.978,A -85,B 0,C 180,E1 -7211.962,E2 -7211.962} C_VEL
LIN {X 0,Y 474.698,Z 273.974,A -85,B 0,C 180,E1 -7215.456,E2 -7215.456} C_VEL
LIN {X 0,Y 474.66,Z 273.978,A -85,B 0,C 180,E1 -7219.01,E2 -7219.01} C_VEL
LIN {X 0,Y 474.588,Z 273.996,A -85,B 0,C 180,E1 -7221.729,E2 -7221.729} C_VEL
LIN {X 0,Y 474.635,Z 273.972,A -85,B 0,C 180,E1 -7224.494,E2 -7224.494} C_VEL
LIN {X 0,Y 474.635,Z 273.981,A -85,B 0,C 180,E1 -7227.324,E2 -7227.324} C_VEL
LIN {X 0,Y 474.601,Z 273.985,A -85,B 0,C 180,E1 -7230.23,E2 -7230.23} C_VEL
LIN {X 0,Y 474.641,Z 273.978,A -85,B 0,C 180,E1 -7233.22,E2 -7233.22} C_VEL
LIN {X 0,Y 474.588,Z 273.986,A -85,B 0,C 180,E1 -7236.323,E2 -7236.323} C_VEL
LIN {X 0,Y 474.626,Z 273.991,A -85,B 0,C 180,E1 -7239.648,E2 -7239.648} C_VEL
LIN {X 0,Y 474.613,Z 273.987,A -85,B 0,C 180,E1 -7242.934,E2 -7242.934} C_VEL
LIN {X 0,Y 474.604,Z 273.991,A -85,B 0,C 180,E1 -7245.895,E2 -7245.895} C_VEL
LIN {X 0,Y 474.626,Z 273.985,A -85,B 0,C 180,E1 -7249.041,E2 -7249.041} C_VEL
LIN {X 0,Y 474.609,Z 273.993,A -85,B 0,C 180,E1 -7251.704,E2 -7251.704} C_VEL
LIN {X 0,Y 474.628,Z 273.988,A -85,B 0,C 180,E1 -7254.726,E2 -7254.726} C_VEL
LIN {X 0,Y 474.634,Z 273.987,A -85,B 0,C 180,E1 -7257.788,E2 -7257.788} C_VEL
LIN {X 0,Y 474.62,Z 274.066,A -85,B 0,C 180,E1 -7259.48,E2 -7259.48} C_VEL
LIN {X 0,Y 477.919,Z 287.434,A -85,B 0,C 180,E1 -7261.69,E2 -7261.69} C_VEL
LIN {X 0,Y 479.225,Z 293.945,A -85,B 0,C 180,E1 -7262.723,E2 -7262.723} C_VEL
LIN {X 0,Y 478.071,Z 315.815,A -85,B 0,C 180,E1 -7265.834,E2 -7265.834} C_VEL
LIN {X 0,Y 477.916,Z 318.523,A -85,B 0,C 180,E1 -7266.216,E2 -7266.216} C_VEL
LIN {X 0,Y 482.436,Z 342.45,A -85,B 0,C 180,E1 -7266.839,E2 -7266.839} C_VEL
LIN {X 0,Y 480.791,Z 485.796,A -85,B 0,C 180,E1 -7269.043,E2 -7269.043} C_VEL
LIN {X 0,Y 480.266,Z 501.47,A -85,B 0,C 180,E1 -7269.459,E2 -7269.459} C_VEL
LIN {X 0,Y 479.638,Z 516.803,A -85,B 0,C 180,E1 -7270.052,E2 -7270.052} C_VEL
LIN {X 0,Y 478.928,Z 530.082,A -85,B 0,C 180,E1 -7270.721,E2 -7270.721} C_VEL
LIN {X 0,Y 478.161,Z 543.609,A -85,B 0,C 180,E1 -7271.579,E2 -7271.579} C_VEL
LIN {X 0,Y 477.365,Z 556.088,A -85,B 0,C 180,E1 -7272.545,E2 -7272.545} C_VEL
LIN {X 0,Y 476.563,Z 568.787,A -85,B 0,C 180,E1 -7273.728,E2 -7273.728} C_VEL
LIN {X 0,Y 475.818,Z 580.329,A -85,B 0,C 180,E1 -7275.02,E2 -7275.02} C_VEL
LIN {X 0,Y 475.241,Z 590.05,A -85,B 0,C 180,E1 -7276.314,E2 -7276.314} C_VEL
LIN {X 0,Y 474.679,Z 599.118,A -85,B 0,C 180,E1 -7277.736,E2 -7277.736} C_VEL
LIN {X 0,Y 474.366,Z 607.565,A -85,B 0,C 180,E1 -7279.328,E2 -7279.328} C_VEL
LIN {X 0,Y 474.018,Z 614.999,A -85,B 0,C 180,E1 -7281.044,E2 -7281.044} C_VEL
LIN {X 0,Y 473.899,Z 620.903,A -85,B 0,C 180,E1 -7282.759,E2 -7282.759} C_VEL
LIN {X 0,Y 473.787,Z 624.41,A -85,B 0,C 180,E1 -7284.04,E2 -7284.04} C_VEL
LIN {X 0,Y 473.703,Z 627.956,A -85,B 0,C 180,E1 -7285.746,E2 -7285.746} C_VEL
LIN {X 0,Y 473.736,Z 630.291,A -85,B 0,C 180,E1 -7287.45,E2 -7287.45} C_VEL
LIN {X 0,Y 473.686,Z 631.464,A -85,B 0,C 180,E1 -7289.15,E2 -7289.15} C_VEL
LIN {X 0,Y 473.686,Z 631.463,A -85,B 0,C 180,E1 -7290.851,E2 -7290.851} C_VEL
LIN {X 0,Y 473.736,Z 630.286,A -85,B 0,C 180,E1 -7292.551,E2 -7292.551} C_VEL
LIN {X 0,Y 473.704,Z 627.95,A -85,B 0,C 180,E1 -7294.255,E2 -7294.255} C_VEL
LIN {X 0,Y 473.78,Z 624.409,A -85,B 0,C 180,E1 -7295.961,E2 -7295.961} C_VEL
LIN {X 0,Y 473.908,Z 619.572,A -85,B 0,C 180,E1 -7297.671,E2 -7297.671} C_VEL
LIN {X 0,Y 474.085,Z 613.307,A -85,B 0,C 180,E1 -7299.385,E2 -7299.385} C_VEL
LIN {X 0,Y 474.489,Z 605.447,A -85,B 0,C 180,E1 -7301.102,E2 -7301.102} C_VEL
LIN {X 0,Y 474.848,Z 596.868,A -85,B 0,C 180,E1 -7302.645,E2 -7302.645} C_VEL
LIN {X 0,Y 475.415,Z 587.019,A -85,B 0,C 180,E1 -7304.118,E2 -7304.118} C_VEL
LIN {X 0,Y 476.038,Z 576.728,A -85,B 0,C 180,E1 -7305.412,E2 -7305.412} C_VEL
LIN {X 0,Y 476.819,Z 564.971,A -85,B 0,C 180,E1 -7306.653,E2 -7306.653} C_VEL
LIN {X 0,Y 477.599,Z 552.182,A -85,B 0,C 180,E1 -7307.779,E2 -7307.779} C_VEL
LIN {X 0,Y 478.455,Z 538.814,A -85,B 0,C 180,E1 -7308.743,E2 -7308.743} C_VEL
LIN {X 0,Y 479.244,Z 524.064,A -85,B 0,C 180,E1 -7309.601,E2 -7309.601} C_VEL
LIN {X 0,Y 479.982,Z 508.205,A -85,B 0,C 180,E1 -7310.306,E2 -7310.306} C_VEL
LIN {X 0,Y 480.604,Z 492.576,A -85,B 0,C 180,E1 -7310.798,E2 -7310.798} C_VEL
LIN {X 0,Y 480.923,Z 476.653,A -85,B 0,C 180,E1 -7311.12,E2 -7311.12} C_VEL
LIN {X 0,Y 482.361,Z 342.292,A -85,B 0,C 180,E1 -7313.166,E2 -7313.166} C_VEL
LIN {X 0,Y 477.919,Z 318.514,A -85,B 0,C 180,E1 -7313.783,E2 -7313.783} C_VEL
LIN {X 0,Y 479.027,Z 298.044,A -85,B 0,C 180,E1 -7316.687,E2 -7316.687} C_VEL
LIN {X 0,Y 479.066,Z 292.292,A -85,B 0,C 180,E1 -7317.524,E2 -7317.524} C_VEL
LIN {X 0,Y 475.126,Z 275.966,A -85,B 0,C 180,E1 -7320.194,E2 -7320.194} C_VEL
LIN {X 0,Y 474.628,Z 273.989,A -85,B 0,C 180,E1 -7320.569,E2 -7320.569} C_VEL
LIN {X 0,Y 474.645,Z 273.987,A -85,B 0,C 180,E1 -7323.22,E2 -7323.22} C_VEL
LIN {X 0,Y 474.591,Z 273.995,A -85,B 0,C 180,E1 -7326.324,E2 -7326.324} C_VEL
LIN {X 0,Y 474.615,Z 273.982,A -85,B 0,C 180,E1 -7329.646,E2 -7329.646} C_VEL
LIN {X 0,Y 474.602,Z 273.992,A -85,B 0,C 180,E1 -7332.234,E2 -7332.234} C_VEL
LIN {X 0,Y 474.619,Z 273.985,A -85,B 0,C 180,E1 -7335.298,E2 -7335.298} C_VEL
LIN {X 0,Y 474.624,Z 273.989,A -85,B 0,C 180,E1 -7338.215,E2 -7338.215} C_VEL
LIN {X 0,Y 474.612,Z 273.987,A -85,B 0,C 180,E1 -7341.543,E2 -7341.543} C_VEL
LIN {X 0,Y 474.625,Z 273.985,A -85,B 0,C 180,E1 -7344.726,E2 -7344.726} C_VEL
LIN {X 0,Y 474.64,Z 273.983,A -85,B 0,C 180,E1 -7347.788,E2 -7347.788} C_VEL
LIN {X 0,Y 474.611,Z 273.984,A -85,B 0,C 180,E1 -7350.889,E2 -7350.889} C_VEL
LIN {X 0,Y 474.608,Z 273.986,A -85,B 0,C 180,E1 -7353.625,E2 -7353.625} C_VEL
LIN {X 0,Y 474.639,Z 273.981,A -85,B 0,C 180,E1 -7356.642,E2 -7356.642} C_VEL
LIN {X 0,Y 474.657,Z 273.985,A -85,B 0,C 180,E1 -7360.09,E2 -7360.09} C_VEL
LIN {X 0,Y 474.639,Z 273.984,A -85,B 0,C 180,E1 -7362.774,E2 -7362.774} C_VEL
LIN {X 0,Y 474.651,Z 273.98,A -85,B 0,C 180,E1 -7365.421,E2 -7365.421} C_VEL
LIN {X 0,Y 474.71,Z 273.977,A -85,B 0,C 180,E1 -7368.038,E2 -7368.038} C_VEL
LIN {X 0,Y 474.701,Z 273.978,A -85,B 0,C 180,E1 -7371.486,E2 -7371.486} C_VEL
LIN {X 0,Y 474.744,Z 273.976,A -85,B 0,C 180,E1 -7374.052,E2 -7374.052} C_VEL
LIN {X 0,Y 474.877,Z 273.953,A -85,B 0,C 180,E1 -7377.455,E2 -7377.455} C_VEL
LIN {X 0,Y 474.884,Z 273.957,A -85,B 0,C 180,E1 -7380,E2 -7380} C_VEL
LIN {X 0,Y 474.886,Z 273.952,A -85,B 0,C 180,E1 -7382.545,E2 -7382.545} C_VEL
LIN {X 0,Y 474.734,Z 273.973,A -85,B 0,C 180,E1 -7385.948,E2 -7385.948} C_VEL
LIN {X 0,Y 474.671,Z 273.979,A -85,B 0,C 180,E1 -7388.515,E2 -7388.515} C_VEL
LIN {X 0,Y 474.709,Z 273.979,A -85,B 0,C 180,E1 -7391.962,E2 -7391.962} C_VEL
LIN {X 0,Y 474.657,Z 273.987,A -85,B 0,C 180,E1 -7395.755,E2 -7395.755} C_VEL
LIN {X 0,Y 474.608,Z 273.985,A -85,B 0,C 180,E1 -7399.013,E2 -7399.013} C_VEL
LIN {X 0,Y 474.579,Z 273.993,A -85,B 0,C 180,E1 -7401.729,E2 -7401.729} C_VEL
LIN {X 0,Y 474.624,Z 273.985,A -85,B 0,C 180,E1 -7404.495,E2 -7404.495} C_VEL
LIN {X 0,Y 474.596,Z 273.984,A -85,B 0,C 180,E1 -7407.327,E2 -7407.327} C_VEL
LIN {X 0,Y 474.553,Z 273.993,A -85,B 0,C 180,E1 -7410.234,E2 -7410.234} C_VEL
LIN {X 0,Y 474.611,Z 273.99,A -85,B 0,C 180,E1 -7413.223,E2 -7413.223} C_VEL
LIN {X 0,Y 474.568,Z 273.99,A -85,B 0,C 180,E1 -7416.326,E2 -7416.326} C_VEL
LIN {X 0,Y 474.599,Z 273.993,A -85,B 0,C 180,E1 -7419.55,E2 -7419.55} C_VEL
LIN {X 0,Y 474.567,Z 273.995,A -85,B 0,C 180,E1 -7422.94,E2 -7422.94} C_VEL
LIN {X 0,Y 474.545,Z 273.995,A -85,B 0,C 180,E1 -7425.887,E2 -7425.887} C_VEL
LIN {X 0,Y 474.581,Z 273.995,A -85,B 0,C 180,E1 -7429.047,E2 -7429.047} C_VEL
LIN {X 0,Y 474.584,Z 273.991,A -85,B 0,C 180,E1 -7431.708,E2 -7431.708} C_VEL
LIN {X 0,Y 474.605,Z 273.992,A -85,B 0,C 180,E1 -7434.723,E2 -7434.723} C_VEL
LIN {X 0,Y 474.612,Z 273.987,A -85,B 0,C 180,E1 -7437.785,E2 -7437.785} C_VEL
LIN {X 0,Y 474.577,Z 273.995,A -85,B 0,C 180,E1 -7440.895,E2 -7440.895} C_VEL
LIN {X 0,Y 474.617,Z 273.993,A -85,B 0,C 180,E1 -7443.921,E2 -7443.921} C_VEL
LIN {X 0,Y 477.384,Z 286.205,A -85,B 0,C 180,E1 -7446.251,E2 -7446.251} C_VEL
LIN {X 0,Y 479.965,Z 293.889,A -85,B 0,C 180,E1 -7446.521,E2 -7446.521} C_VEL
